LIN {X 95.616,Y 104.988,Z 83.161,A 180.000,B 0.000,C 180.000} C_DIS
LIN {X 95.371,Y 104.988,Z 83.026,A 180.000,B 0.000,C 180.000} C_DIS
LIN {X 94.812,Y 104.988,Z 82.658,A 180.000,B 0.000,C 180.000} C_DIS
LIN {X 94.419,Y 104.988,Z 82.358,A 180.000,B 0.000,C 180.000} C_DIS
LIN {X 93.998,Y 104.988,Z 81.987,A 180.000,B 0.000,C 180.000} C_DIS
LIN {X 93.703,Y 104.988,Z 81.713,A 180.000,B 0.000,C 180.000} C_DIS
LIN {X 93.333,Y 104.988,Z 81.344,A 180.000,B 0.000,C 180.000} C_DIS
LIN {X 92.872,Y 104.988,Z 80.840,A 180.000,B 0.000,C 180.000} C_DIS
LIN {X 92.497,Y 104.988,Z 80.403,A 180.000,B 0.000,C 180.000} C_DIS
LIN {X 92.120,Y 104.988,Z 79.949,A 180.000,B 0.000,C 180.000} C_DIS
LIN {X 91.570,Y 104.988,Z 79.235,A 180.000,B 0.000,C 180.000} C_DIS
LIN {X 90.776,Y 104.988,Z 78.140,A 180.000,B 0.000,C 180.000} C_DIS
LIN {X 90.026,Y 104.988,Z 77.033,A 180.000,B 0.000,C 180.000} C_DIS
LIN {X 89.022,Y 104.988,Z 75.463,A 180.000,B 0.000,C 180.000} C_DIS
LIN {X 88.077,Y 104.988,Z 73.911,A 180.000,B 0.000,C 180.000} C_DIS
LIN {X 86.884,Y 104.988,Z 71.862,A 180.000,B 0.000,C 180.000} C_DIS
LIN {X 85.520,Y 104.988,Z 69.426,A 180.000,B 0.000,C 180.000} C_DIS
LIN {X 84.508,Y 104.988,Z 67.555,A 180.000,B 0.000,C 180.000} C_DIS
LIN {X 84.508,Y 104.988,Z 62.000,A 180.000,B 0.000,C 180.000} C_DIS
LIN {X 70.550,Y 104.988,Z 62.000,A 180.000,B 0.000,C 180.000} C_DIS
LIN {X 70.550,Y 104.988,Z 66.500,A 180.000,B 0.000,C 180.000} C_DIS
LIN {X 70.498,Y 104.988,Z 66.500,A 180.000,B 0.000,C 180.000} C_DIS
LIN {X 70.498,Y 104.988,Z 70.000,A 180.000,B 0.000,C 180.000} C_DIS
LIN {X 65.196,Y 104.988,Z 70.000,A 180.000,B 0.000,C 180.000} C_DIS
LIN {X 65.195,Y 104.988,Z 74.500,A 180.000,B 0.000,C 180.000} C_DIS
LIN {X 65.139,Y 104.988,Z 74.500,A 180.000,B 0.000,C 180.000} C_DIS
LIN {X 65.139,Y 104.988,Z 78.000,A 180.000,B 0.000,C 180.000} C_DIS
LIN {X 51.866,Y 104.988,Z 78.000,A 180.000,B 0.000,C 180.000} C_DIS
LIN {X 51.866,Y 104.988,Z 74.500,A 180.000,B 0.000,C 180.000} C_DIS
LIN {X 51.810,Y 104.988,Z 74.500,A 180.000,B 0.000,C 180.000} C_DIS
LIN {X 51.809,Y 104.988,Z 70.000,A 180.000,B 0.000,C 180.000} C_DIS
LIN {X 46.502,Y 104.988,Z 70.000,A 180.000,B 0.000,C 180.000} C_DIS
LIN {X 46.499,Y 104.988,Z 66.500,A 180.000,B 0.000,C 180.000} C_DIS
LIN {X 46.450,Y 104.988,Z 66.500,A 180.000,B 0.000,C 180.000} C_DIS
LIN {X 46.450,Y 104.988,Z 62.000,A 180.000,B 0.000,C 180.000} C_DIS
LIN {X 36.453,Y 104.988,Z 62.000,A 180.000,B 0.000,C 180.000} C_DIS
LIN {X 36.453,Y 104.988,Z 57.000,A 180.000,B 0.000,C 180.000} C_DIS
LIN {X 7.719,Y 104.988,Z 57.000,A 180.000,B 0.000,C 180.000} C_DIS
LIN {X 7.719,Y 104.988,Z 52.000,A 180.000,B 0.000,C 180.000} C_DIS
LIN {X 2.500,Y 104.988,Z 52.000,A 180.000,B 0.000,C 180.000} C_DIS
LIN {X 2.500,Y 104.988,Z 45.000,A 180.000,B 0.000,C 180.000} C_DIS
LIN {X -0.010,Y 104.988,Z 45.000,A 180.000,B 0.000,C 180.000} C_DIS
; Link Move Starts
LIN {X -0.120,Y 104.988,Z 45.026,A 180.000,B 0.000,C 180.000} C_DIS
LIN {X -0.230,Y 104.988,Z 45.051,A 180.000,B 0.000,C 180.000} C_DIS
LIN {X -0.771,Y 105.301,Z 45.051,A 180.000,B 0.000,C 180.000} C_DIS
LIN {X -0.771,Y 105.926,Z 45.051,A 180.000,B 0.000,C 180.000} C_DIS
LIN {X -0.230,Y 106.238,Z 45.051,A 180.000,B 0.000,C 180.000} C_DIS
LIN {X -0.120,Y 106.238,Z 45.026,A 180.000,B 0.000,C 180.000} C_DIS
LIN {X -0.010,Y 106.238,Z 45.000,A 180.000,B 0.000,C 180.000} C_DIS
; Cutting Move Starts
LIN {X 2.500,Y 106.238,Z 45.000,A 180.000,B 0.000,C 180.000} C_DIS
LIN {X 2.500,Y 106.238,Z 52.000,A 180.000,B 0.000,C 180.000} C_DIS
LIN {X 8.224,Y 106.238,Z 52.000,A 180.000,B 0.000,C 180.000} C_DIS
LIN {X 8.228,Y 106.238,Z 57.000,A 180.000,B 0.000,C 180.000} C_DIS
LIN {X 37.703,Y 106.238,Z 57.000,A 180.000,B 0.000,C 180.000} C_DIS
LIN {X 37.703,Y 106.238,Z 62.000,A 180.000,B 0.000,C 180.000} C_DIS
LIN {X 46.881,Y 106.238,Z 62.000,A 180.000,B 0.000,C 180.000} C_DIS
LIN {X 46.881,Y 106.238,Z 66.500,A 180.000,B 0.000,C 180.000} C_DIS
LIN {X 46.935,Y 106.238,Z 66.500,A 180.000,B 0.000,C 180.000} C_DIS
LIN {X 46.936,Y 106.238,Z 70.000,A 180.000,B 0.000,C 180.000} C_DIS
LIN {X 52.627,Y 106.238,Z 70.000,A 180.000,B 0.000,C 180.000} C_DIS
LIN {X 52.627,Y 106.238,Z 74.500,A 180.000,B 0.000,C 180.000} C_DIS
LIN {X 52.691,Y 106.238,Z 74.500,A 180.000,B 0.000,C 180.000} C_DIS
LIN {X 52.691,Y 106.238,Z 78.000,A 180.000,B 0.000,C 180.000} C_DIS
LIN {X 64.310,Y 106.238,Z 78.000,A 180.000,B 0.000,C 180.000} C_DIS
LIN {X 64.310,Y 106.238,Z 74.500,A 180.000,B 0.000,C 180.000} C_DIS
LIN {X 64.371,Y 106.238,Z 74.500,A 180.000,B 0.000,C 180.000} C_DIS
LIN {X 64.376,Y 106.238,Z 70.000,A 180.000,B 0.000,C 180.000} C_DIS
LIN {X 70.063,Y 106.238,Z 70.000,A 180.000,B 0.000,C 180.000} C_DIS
LIN {X 70.064,Y 106.238,Z 66.500,A 180.000,B 0.000,C 180.000} C_DIS
LIN {X 70.119,Y 106.238,Z 66.500,A 180.000,B 0.000,C 180.000} C_DIS
LIN {X 70.119,Y 106.238,Z 62.000,A 180.000,B 0.000,C 180.000} C_DIS
LIN {X 85.309,Y 106.238,Z 62.000,A 180.000,B 0.000,C 180.000} C_DIS
LIN {X 85.309,Y 106.238,Z 67.555,A 180.000,B 0.000,C 180.000} C_DIS
LIN {X 86.499,Y 106.238,Z 69.593,A 180.000,B 0.000,C 180.000} C_DIS
LIN {X 87.652,Y 106.238,Z 71.487,A 180.000,B 0.000,C 180.000} C_DIS
LIN {X 88.751,Y 106.238,Z 73.204,A 180.000,B 0.000,C 180.000} C_DIS
LIN {X 89.638,Y 106.238,Z 74.514,A 180.000,B 0.000,C 180.000} C_DIS
LIN {X 90.553,Y 106.238,Z 75.781,A 180.000,B 0.000,C 180.000} C_DIS
LIN {X 91.246,Y 106.238,Z 76.678,A 180.000,B 0.000,C 180.000} C_DIS
LIN {X 91.704,Y 106.238,Z 77.229,A 180.000,B 0.000,C 180.000} C_DIS
LIN {X 92.068,Y 106.238,Z 77.653,A 180.000,B 0.000,C 180.000} C_DIS
LIN {X 92.647,Y 106.238,Z 78.287,A 180.000,B 0.000,C 180.000} C_DIS
LIN {X 93.102,Y 106.238,Z 78.739,A 180.000,B 0.000,C 180.000} C_DIS
LIN {X 93.353,Y 106.238,Z 78.974,A 180.000,B 0.000,C 180.000} C_DIS
LIN {X 93.850,Y 106.238,Z 79.413,A 180.000,B 0.000,C 180.000} C_DIS
LIN {X 94.082,Y 106.238,Z 79.596,A 180.000,B 0.000,C 180.000} C_DIS
LIN {X 94.407,Y 106.238,Z 79.842,A 180.000,B 0.000,C 180.000} C_DIS
LIN {X 95.017,Y 106.238,Z 80.240,A 180.000,B 0.000,C 180.000} C_DIS
LIN {X 95.429,Y 106.238,Z 80.463,A 180.000,B 0.000,C 180.000} C_DIS
LIN {X 95.636,Y 106.238,Z 80.555,A 180.000,B 0.000,C 180.000} C_DIS
LIN {X 96.080,Y 106.238,Z 80.735,A 180.000,B 0.000,C 180.000} C_DIS
LIN {X 96.484,Y 106.238,Z 80.857,A 180.000,B 0.000,C 180.000} C_DIS
LIN {X 96.776,Y 106.238,Z 80.912,A 180.000,B 0.000,C 180.000} C_DIS
LIN {X 97.029,Y 106.238,Z 80.950,A 180.000,B 0.000,C 180.000} C_DIS
LIN {X 97.255,Y 106.238,Z 80.971,A 180.000,B 0.000,C 180.000} C_DIS
LIN {X 97.526,Y 106.238,Z 80.983,A 180.000,B 0.000,C 180.000} C_DIS
LIN {X 97.834,Y 106.238,Z 80.966,A 180.000,B 0.000,C 180.000} C_DIS
LIN {X 98.107,Y 106.238,Z 80.932,A 180.000,B 0.000,C 180.000} C_DIS
LIN {X 98.493,Y 106.238,Z 80.862,A 180.000,B 0.000,C 180.000} C_DIS
LIN {X 98.803,Y 106.238,Z 80.772,A 180.000,B 0.000,C 180.000} C_DIS
LIN {X 98.999,Y 106.238,Z 80.704,A 180.000,B 0.000,C 180.000} C_DIS
LIN {X 99.513,Y 106.238,Z 80.491,A 180.000,B 0.000,C 180.000} C_DIS
LIN {X 99.761,Y 106.238,Z 80.362,A 180.000,B 0.000,C 180.000} C_DIS
LIN {X 100.001,Y 106.238,Z 80.229,A 180.000,B 0.000,C 180.000} C_DIS
LIN {X 100.606,Y 106.238,Z 79.832,A 180.000,B 0.000,C 180.000} C_DIS
LIN {X 101.068,Y 106.238,Z 79.481,A 180.000,B 0.000,C 180.000} C_DIS
LIN {X 101.407,Y 106.238,Z 79.188,A 180.000,B 0.000,C 180.000} C_DIS
LIN {X 101.768,Y 106.238,Z 78.864,A 180.000,B 0.000,C 180.000} C_DIS
LIN {X 102.297,Y 106.238,Z 78.345,A 180.000,B 0.000,C 180.000} C_DIS
LIN {X 102.749,Y 106.238,Z 77.856,A 180.000,B 0.000,C 180.000} C_DIS
LIN {X 103.049,Y 106.238,Z 77.520,A 180.000,B 0.000,C 180.000} C_DIS
LIN {X 103.690,Y 106.238,Z 76.757,A 180.000,B 0.000,C 180.000} C_DIS
LIN {X 104.418,Y 106.238,Z 75.820,A 180.000,B 0.000,C 180.000} C_DIS
LIN {X 105.298,Y 106.238,Z 74.605,A 180.000,B 0.000,C 180.000} C_DIS
LIN {X 106.168,Y 106.238,Z 73.327,A 180.000,B 0.000,C 180.000} C_DIS
LIN {X 107.258,Y 106.238,Z 71.631,A 180.000,B 0.000,C 180.000} C_DIS
LIN {X 108.395,Y 106.238,Z 69.771,A 180.000,B 0.000,C 180.000} C_DIS
LIN {X 109.689,Y 106.238,Z 67.558,A 180.000,B 0.000,C 180.000} C_DIS
LIN {X 109.691,Y 106.238,Z 62.000,A 180.000,B 0.000,C 180.000} C_DIS
LIN {X 117.295,Y 106.238,Z 62.000,A 180.000,B 0.000,C 180.000} C_DIS
LIN {X 117.297,Y 106.238,Z 57.000,A 180.000,B 0.000,C 180.000} C_DIS
LIN {X 146.772,Y 106.238,Z 57.000,A 180.000,B 0.000,C 180.000} C_DIS
LIN {X 146.772,Y 106.238,Z 52.000,A 180.000,B 0.000,C 180.000} C_DIS
LIN {X 152.500,Y 106.238,Z 52.000,A 180.000,B 0.000,C 180.000} C_DIS
LIN {X 152.500,Y 106.238,Z 45.000,A 180.000,B 0.000,C 180.000} C_DIS
LIN {X 155.010,Y 106.238,Z 45.000,A 180.000,B 0.000,C 180.000} C_DIS
; Link Move Starts
LIN {X 155.120,Y 106.238,Z 45.026,A 180.000,B 0.000,C 180.000} C_DIS
LIN {X 155.230,Y 106.238,Z 45.051,A 180.000,B 0.000,C 180.000} C_DIS
LIN {X 155.771,Y 106.551,Z 45.051,A 180.000,B 0.000,C 180.000} C_DIS
LIN {X 155.771,Y 107.176,Z 45.051,A 180.000,B 0.000,C 180.000} C_DIS
LIN {X 155.230,Y 107.488,Z 45.051,A 180.000,B 0.000,C 180.000} C_DIS
LIN {X 155.120,Y 107.488,Z 45.026,A 180.000,B 0.000,C 180.000} C_DIS
LIN {X 155.010,Y 107.488,Z 45.000,A 180.000,B 0.000,C 180.000} C_DIS
; Cutting Move Starts
LIN {X 152.500,Y 107.488,Z 45.000,A 180.000,B 0.000,C 180.000} C_DIS
LIN {X 152.500,Y 107.488,Z 52.000,A 180.000,B 0.000,C 180.000} C_DIS
LIN {X 146.238,Y 107.488,Z 52.000,A 180.000,B 0.000,C 180.000} C_DIS
LIN {X 146.238,Y 107.488,Z 57.000,A 180.000,B 0.000,C 180.000} C_DIS
LIN {X 116.047,Y 107.488,Z 57.000,A 180.000,B 0.000,C 180.000} C_DIS
LIN {X 116.047,Y 107.488,Z 62.000,A 180.000,B 0.000,C 180.000} C_DIS
LIN {X 108.691,Y 107.488,Z 62.000,A 180.000,B 0.000,C 180.000} C_DIS
LIN {X 108.688,Y 107.488,Z 67.559,A 180.000,B 0.000,C 180.000} C_DIS
LIN {X 107.443,Y 107.488,Z 69.499,A 180.000,B 0.000,C 180.000} C_DIS
LIN {X 106.403,Y 107.488,Z 71.028,A 180.000,B 0.000,C 180.000} C_DIS
LIN {X 105.423,Y 107.488,Z 72.382,A 180.000,B 0.000,C 180.000} C_DIS
LIN {X 104.570,Y 107.488,Z 73.479,A 180.000,B 0.000,C 180.000} C_DIS
LIN {X 103.804,Y 107.488,Z 74.390,A 180.000,B 0.000,C 180.000} C_DIS
LIN {X 103.504,Y 107.488,Z 74.725,A 180.000,B 0.000,C 180.000} C_DIS
LIN {X 102.991,Y 107.488,Z 75.279,A 180.000,B 0.000,C 180.000} C_DIS
LIN {X 102.351,Y 107.488,Z 75.907,A 180.000,B 0.000,C 180.000} C_DIS
LIN {X 102.000,Y 107.488,Z 76.221,A 180.000,B 0.000,C 180.000} C_DIS
LIN {X 101.597,Y 107.488,Z 76.571,A 180.000,B 0.000,C 180.000} C_DIS
LIN {X 101.032,Y 107.488,Z 77.002,A 180.000,B 0.000,C 180.000} C_DIS
LIN {X 100.369,Y 107.488,Z 77.435,A 180.000,B 0.000,C 180.000} C_DIS
LIN {X 100.126,Y 107.488,Z 77.570,A 180.000,B 0.000,C 180.000} C_DIS
LIN {X 99.798,Y 107.488,Z 77.742,A 180.000,B 0.000,C 180.000} C_DIS
LIN {X 99.210,Y 107.488,Z 77.987,A 180.000,B 0.000,C 180.000} C_DIS
LIN {X 99.019,Y 107.488,Z 78.052,A 180.000,B 0.000,C 180.000} C_DIS
LIN {X 98.633,Y 107.488,Z 78.165,A 180.000,B 0.000,C 180.000} C_DIS
LIN {X 98.157,Y 107.488,Z 78.251,A 180.000,B 0.000,C 180.000} C_DIS
LIN {X 97.920,Y 107.488,Z 78.280,A 180.000,B 0.000,C 180.000} C_DIS
LIN {X 97.529,Y 107.488,Z 78.303,A 180.000,B 0.000,C 180.000} C_DIS
LIN {X 97.268,Y 107.488,Z 78.291,A 180.000,B 0.000,C 180.000} C_DIS
LIN {X 96.984,Y 107.488,Z 78.270,A 180.000,B 0.000,C 180.000} C_DIS
LIN {X 96.715,Y 107.488,Z 78.230,A 180.000,B 0.000,C 180.000} C_DIS
LIN {X 96.353,Y 107.488,Z 78.162,A 180.000,B 0.000,C 180.000} C_DIS
LIN {X 95.857,Y 107.488,Z 78.013,A 180.000,B 0.000,C 180.000} C_DIS
LIN {X 95.438,Y 107.488,Z 77.842,A 180.000,B 0.000,C 180.000} C_DIS
LIN {X 95.169,Y 107.488,Z 77.727,A 180.000,B 0.000,C 180.000} C_DIS
LIN {X 94.651,Y 107.488,Z 77.448,A 180.000,B 0.000,C 180.000} C_DIS
LIN {X 93.979,Y 107.488,Z 77.009,A 180.000,B 0.000,C 180.000} C_DIS
LIN {X 93.591,Y 107.488,Z 76.716,A 180.000,B 0.000,C 180.000} C_DIS
LIN {X 93.340,Y 107.488,Z 76.518,A 180.000,B 0.000,C 180.000} C_DIS
LIN {X 92.731,Y 107.488,Z 75.982,A 180.000,B 0.000,C 180.000} C_DIS
LIN {X 92.465,Y 107.488,Z 75.730,A 180.000,B 0.000,C 180.000} C_DIS
LIN {X 91.957,Y 107.488,Z 75.226,A 180.000,B 0.000,C 180.000} C_DIS
LIN {X 91.256,Y 107.488,Z 74.459,A 180.000,B 0.000,C 180.000} C_DIS
LIN {X 90.882,Y 107.488,Z 74.020,A 180.000,B 0.000,C 180.000} C_DIS
LIN {X 90.370,Y 107.488,Z 73.405,A 180.000,B 0.000,C 180.000} C_DIS
LIN {X 89.537,Y 107.488,Z 72.327,A 180.000,B 0.000,C 180.000} C_DIS
LIN {X 88.532,Y 107.488,Z 70.935,A 180.000,B 0.000,C 180.000} C_DIS
LIN {X 87.483,Y 107.488,Z 69.386,A 180.000,B 0.000,C 180.000} C_DIS
LIN {X 86.309,Y 107.488,Z 67.555,A 180.000,B 0.000,C 180.000} C_DIS
LIN {X 86.308,Y 107.488,Z 62.000,A 180.000,B 0.000,C 180.000} C_DIS
LIN {X 69.529,Y 107.488,Z 62.000,A 180.000,B 0.000,C 180.000} C_DIS
LIN {X 69.528,Y 107.488,Z 66.500,A 180.000,B 0.000,C 180.000} C_DIS
LIN {X 69.472,Y 107.488,Z 66.500,A 180.000,B 0.000,C 180.000} C_DIS
LIN {X 69.471,Y 107.488,Z 70.000,A 180.000,B 0.000,C 180.000} C_DIS
LIN {X 63.096,Y 107.488,Z 70.000,A 180.000,B 0.000,C 180.000} C_DIS
LIN {X 63.096,Y 107.488,Z 74.500,A 180.000,B 0.000,C 180.000} C_DIS
LIN {X 63.016,Y 107.488,Z 74.500,A 180.000,B 0.000,C 180.000} C_DIS
LIN {X 63.014,Y 107.488,Z 78.000,A 180.000,B 0.000,C 180.000} C_DIS
LIN {X 53.992,Y 107.488,Z 78.000,A 180.000,B 0.000,C 180.000} C_DIS
LIN {X 53.992,Y 107.488,Z 74.500,A 180.000,B 0.000,C 180.000} C_DIS
LIN {X 53.909,Y 107.488,Z 74.500,A 180.000,B 0.000,C 180.000} C_DIS
LIN {X 53.909,Y 107.488,Z 70.000,A 180.000,B 0.000,C 180.000} C_DIS
LIN {X 47.528,Y 107.488,Z 70.000,A 180.000,B 0.000,C 180.000} C_DIS
LIN {X 47.527,Y 107.488,Z 66.500,A 180.000,B 0.000,C 180.000} C_DIS
LIN {X 47.471,Y 107.488,Z 66.500,A 180.000,B 0.000,C 180.000} C_DIS
LIN {X 47.471,Y 107.488,Z 62.000,A 180.000,B 0.000,C 180.000} C_DIS
LIN {X 38.953,Y 107.488,Z 62.000,A 180.000,B 0.000,C 180.000} C_DIS
LIN {X 38.952,Y 107.488,Z 57.000,A 180.000,B 0.000,C 180.000} C_DIS
LIN {X 8.762,Y 107.488,Z 57.000,A 180.000,B 0.000,C 180.000} C_DIS
LIN {X 8.762,Y 107.488,Z 52.000,A 180.000,B 0.000,C 180.000} C_DIS
LIN {X 2.500,Y 107.488,Z 52.000,A 180.000,B 0.000,C 180.000} C_DIS
LIN {X 2.500,Y 107.488,Z 45.000,A 180.000,B 0.000,C 180.000} C_DIS
LIN {X -0.010,Y 107.488,Z 45.000,A 180.000,B 0.000,C 180.000} C_DIS
; Link Move Starts
LIN {X -0.120,Y 107.488,Z 45.026,A 180.000,B 0.000,C 180.000} C_DIS
LIN {X -0.230,Y 107.488,Z 45.051,A 180.000,B 0.000,C 180.000} C_DIS
LIN {X -0.771,Y 107.801,Z 45.051,A 180.000,B 0.000,C 180.000} C_DIS
LIN {X -0.771,Y 108.425,Z 45.051,A 180.000,B 0.000,C 180.000} C_DIS
LIN {X -0.230,Y 108.738,Z 45.051,A 180.000,B 0.000,C 180.000} C_DIS
LIN {X -0.120,Y 108.738,Z 45.026,A 180.000,B 0.000,C 180.000} C_DIS
LIN {X -0.010,Y 108.738,Z 45.000,A 180.000,B 0.000,C 180.000} C_DIS
; Cutting Move Starts
LIN {X 2.500,Y 108.738,Z 45.000,A 180.000,B 0.000,C 180.000} C_DIS
LIN {X 2.500,Y 108.738,Z 52.000,A 180.000,B 0.000,C 180.000} C_DIS
LIN {X 9.316,Y 108.738,Z 52.000,A 180.000,B 0.000,C 180.000} C_DIS
LIN {X 9.320,Y 108.738,Z 57.000,A 180.000,B 0.000,C 180.000} C_DIS
LIN {X 40.202,Y 108.738,Z 57.000,A 180.000,B 0.000,C 180.000} C_DIS
LIN {X 40.202,Y 108.738,Z 62.000,A 180.000,B 0.000,C 180.000} C_DIS
LIN {X 48.247,Y 108.738,Z 62.000,A 180.000,B 0.000,C 180.000} C_DIS
LIN {X 48.251,Y 108.738,Z 66.500,A 180.000,B 0.000,C 180.000} C_DIS
LIN {X 48.311,Y 108.738,Z 66.500,A 180.000,B 0.000,C 180.000} C_DIS
LIN {X 48.311,Y 108.738,Z 70.000,A 180.000,B 0.000,C 180.000} C_DIS
LIN {X 56.369,Y 108.738,Z 70.000,A 180.000,B 0.000,C 180.000} C_DIS
LIN {X 56.369,Y 108.738,Z 74.500,A 180.000,B 0.000,C 180.000} C_DIS
LIN {X 56.545,Y 108.738,Z 74.500,A 180.000,B 0.000,C 180.000} C_DIS
LIN {X 56.545,Y 108.738,Z 78.000,A 180.000,B 0.000,C 180.000} C_DIS
LIN {X 60.452,Y 108.738,Z 78.000,A 180.000,B 0.000,C 180.000} C_DIS
LIN {X 60.452,Y 108.738,Z 74.500,A 180.000,B 0.000,C 180.000} C_DIS
LIN {X 60.648,Y 108.738,Z 74.500,A 180.000,B 0.000,C 180.000} C_DIS
LIN {X 60.648,Y 108.738,Z 70.000,A 180.000,B 0.000,C 180.000} C_DIS
LIN {X 68.685,Y 108.738,Z 70.000,A 180.000,B 0.000,C 180.000} C_DIS
LIN {X 68.689,Y 108.738,Z 66.500,A 180.000,B 0.000,C 180.000} C_DIS
LIN {X 68.749,Y 108.738,Z 66.500,A 180.000,B 0.000,C 180.000} C_DIS
LIN {X 68.749,Y 108.738,Z 62.000,A 180.000,B 0.000,C 180.000} C_DIS
LIN {X 87.566,Y 108.738,Z 62.000,A 180.000,B 0.000,C 180.000} C_DIS
LIN {X 87.566,Y 108.738,Z 67.555,A 180.000,B 0.000,C 180.000} C_DIS
LIN {X 88.517,Y 108.738,Z 68.869,A 180.000,B 0.000,C 180.000} C_DIS
LIN {X 89.472,Y 108.738,Z 70.105,A 180.000,B 0.000,C 180.000} C_DIS
LIN {X 89.816,Y 108.738,Z 70.520,A 180.000,B 0.000,C 180.000} C_DIS
LIN {X 90.450,Y 108.738,Z 71.272,A 180.000,B 0.000,C 180.000} C_DIS
LIN {X 91.276,Y 108.738,Z 72.173,A 180.000,B 0.000,C 180.000} C_DIS
LIN {X 92.056,Y 108.738,Z 72.942,A 180.000,B 0.000,C 180.000} C_DIS
LIN {X 92.410,Y 108.738,Z 73.257,A 180.000,B 0.000,C 180.000} C_DIS
LIN {X 92.879,Y 108.738,Z 73.664,A 180.000,B 0.000,C 180.000} C_DIS
LIN {X 93.546,Y 108.738,Z 74.173,A 180.000,B 0.000,C 180.000} C_DIS
LIN {X 94.282,Y 108.738,Z 74.653,A 180.000,B 0.000,C 180.000} C_DIS
LIN {X 94.896,Y 108.738,Z 74.984,A 180.000,B 0.000,C 180.000} C_DIS
LIN {X 95.231,Y 108.738,Z 75.127,A 180.000,B 0.000,C 180.000} C_DIS
LIN {X 95.631,Y 108.738,Z 75.290,A 180.000,B 0.000,C 180.000} C_DIS
LIN {X 96.220,Y 108.738,Z 75.467,A 180.000,B 0.000,C 180.000} C_DIS
LIN {X 96.675,Y 108.738,Z 75.551,A 180.000,B 0.000,C 180.000} C_DIS
LIN {X 96.914,Y 108.738,Z 75.587,A 180.000,B 0.000,C 180.000} C_DIS
LIN {X 97.296,Y 108.738,Z 75.613,A 180.000,B 0.000,C 180.000} C_DIS
LIN {X 97.537,Y 108.738,Z 75.622,A 180.000,B 0.000,C 180.000} C_DIS
LIN {X 98.004,Y 108.738,Z 75.594,A 180.000,B 0.000,C 180.000} C_DIS
LIN {X 98.208,Y 108.738,Z 75.571,A 180.000,B 0.000,C 180.000} C_DIS
LIN {X 98.773,Y 108.738,Z 75.468,A 180.000,B 0.000,C 180.000} C_DIS
LIN {X 99.123,Y 108.738,Z 75.366,A 180.000,B 0.000,C 180.000} C_DIS
LIN {X 99.388,Y 108.738,Z 75.283,A 180.000,B 0.000,C 180.000} C_DIS
LIN {X 99.965,Y 108.738,Z 75.045,A 180.000,B 0.000,C 180.000} C_DIS
LIN {X 100.174,Y 108.738,Z 74.947,A 180.000,B 0.000,C 180.000} C_DIS
LIN {X 100.723,Y 108.738,Z 74.650,A 180.000,B 0.000,C 180.000} C_DIS
LIN {X 101.455,Y 108.738,Z 74.173,A 180.000,B 0.000,C 180.000} C_DIS
LIN {X 102.121,Y 108.738,Z 73.664,A 180.000,B 0.000,C 180.000} C_DIS
LIN {X 102.549,Y 108.738,Z 73.293,A 180.000,B 0.000,C 180.000} C_DIS
LIN {X 102.932,Y 108.738,Z 72.953,A 180.000,B 0.000,C 180.000} C_DIS
LIN {X 103.673,Y 108.738,Z 72.226,A 180.000,B 0.000,C 180.000} C_DIS
LIN {X 104.030,Y 108.738,Z 71.841,A 180.000,B 0.000,C 180.000} C_DIS
LIN {X 104.563,Y 108.738,Z 71.256,A 180.000,B 0.000,C 180.000} C_DIS
LIN {X 105.451,Y 108.738,Z 70.201,A 180.000,B 0.000,C 180.000} C_DIS
LIN {X 106.426,Y 108.738,Z 68.945,A 180.000,B 0.000,C 180.000} C_DIS
LIN {X 107.434,Y 108.738,Z 67.555,A 180.000,B 0.000,C 180.000} C_DIS
LIN {X 107.434,Y 108.738,Z 62.000,A 180.000,B 0.000,C 180.000} C_DIS
LIN {X 114.795,Y 108.738,Z 62.000,A 180.000,B 0.000,C 180.000} C_DIS
LIN {X 114.798,Y 108.738,Z 57.000,A 180.000,B 0.000,C 180.000} C_DIS
LIN {X 145.680,Y 108.738,Z 57.000,A 180.000,B 0.000,C 180.000} C_DIS
LIN {X 145.680,Y 108.738,Z 52.000,A 180.000,B 0.000,C 180.000} C_DIS
LIN {X 152.500,Y 108.738,Z 52.000,A 180.000,B 0.000,C 180.000} C_DIS
LIN {X 152.500,Y 108.738,Z 45.000,A 180.000,B 0.000,C 180.000} C_DIS
LIN {X 155.010,Y 108.738,Z 45.000,A 180.000,B 0.000,C 180.000} C_DIS
; Link Move Starts
LIN {X 155.120,Y 108.738,Z 45.026,A 180.000,B 0.000,C 180.000} C_DIS
LIN {X 155.230,Y 108.738,Z 45.051,A 180.000,B 0.000,C 180.000} C_DIS
LIN {X 155.771,Y 109.050,Z 45.051,A 180.000,B 0.000,C 180.000} C_DIS
LIN {X 155.771,Y 109.675,Z 45.051,A 180.000,B 0.000,C 180.000} C_DIS
LIN {X 155.230,Y 109.988,Z 45.051,A 180.000,B 0.000,C 180.000} C_DIS
LIN {X 155.120,Y 109.988,Z 45.026,A 180.000,B 0.000,C 180.000} C_DIS
LIN {X 155.010,Y 109.988,Z 45.000,A 180.000,B 0.000,C 180.000} C_DIS
; Cutting Move Starts
LIN {X 152.500,Y 109.988,Z 45.000,A 180.000,B 0.000,C 180.000} C_DIS
LIN {X 152.500,Y 109.988,Z 52.000,A 180.000,B 0.000,C 180.000} C_DIS
LIN {X 145.096,Y 109.988,Z 52.000,A 180.000,B 0.000,C 180.000} C_DIS
LIN {X 145.093,Y 109.988,Z 57.000,A 180.000,B 0.000,C 180.000} C_DIS
LIN {X 113.548,Y 109.988,Z 57.000,A 180.000,B 0.000,C 180.000} C_DIS
LIN {X 113.548,Y 109.988,Z 62.000,A 180.000,B 0.000,C 180.000} C_DIS
LIN {X 105.801,Y 109.988,Z 62.000,A 180.000,B 0.000,C 180.000} C_DIS
LIN {X 105.801,Y 109.988,Z 67.555,A 180.000,B 0.000,C 180.000} C_DIS
LIN {X 105.313,Y 109.988,Z 68.132,A 180.000,B 0.000,C 180.000} C_DIS
LIN {X 104.382,Y 109.988,Z 69.144,A 180.000,B 0.000,C 180.000} C_DIS
LIN {X 103.516,Y 109.988,Z 69.996,A 180.000,B 0.000,C 180.000} C_DIS
LIN {X 102.669,Y 109.988,Z 70.739,A 180.000,B 0.000,C 180.000} C_DIS
LIN {X 101.880,Y 109.988,Z 71.342,A 180.000,B 0.000,C 180.000} C_DIS
LIN {X 101.078,Y 109.988,Z 71.864,A 180.000,B 0.000,C 180.000} C_DIS
LIN {X 100.362,Y 109.988,Z 72.248,A 180.000,B 0.000,C 180.000} C_DIS
LIN {X 99.619,Y 109.988,Z 72.558,A 180.000,B 0.000,C 180.000} C_DIS
LIN {X 99.375,Y 109.988,Z 72.635,A 180.000,B 0.000,C 180.000} C_DIS
LIN {X 98.908,Y 109.988,Z 72.772,A 180.000,B 0.000,C 180.000} C_DIS
LIN {X 98.249,Y 109.988,Z 72.891,A 180.000,B 0.000,C 180.000} C_DIS
LIN {X 98.010,Y 109.988,Z 72.914,A 180.000,B 0.000,C 180.000} C_DIS
LIN {X 97.520,Y 109.988,Z 72.942,A 180.000,B 0.000,C 180.000} C_DIS
LIN {X 97.112,Y 109.988,Z 72.921,A 180.000,B 0.000,C 180.000} C_DIS
LIN {X 96.821,Y 109.988,Z 72.901,A 180.000,B 0.000,C 180.000} C_DIS
LIN {X 96.564,Y 109.988,Z 72.859,A 180.000,B 0.000,C 180.000} C_DIS
LIN {X 96.079,Y 109.988,Z 72.769,A 180.000,B 0.000,C 180.000} C_DIS
LIN {X 95.404,Y 109.988,Z 72.566,A 180.000,B 0.000,C 180.000} C_DIS
LIN {X 94.956,Y 109.988,Z 72.383,A 180.000,B 0.000,C 180.000} C_DIS
LIN {X 94.621,Y 109.988,Z 72.240,A 180.000,B 0.000,C 180.000} C_DIS
LIN {X 93.913,Y 109.988,Z 71.859,A 180.000,B 0.000,C 180.000} C_DIS
LIN {X 93.117,Y 109.988,Z 71.340,A 180.000,B 0.000,C 180.000} C_DIS
LIN {X 92.327,Y 109.988,Z 70.735,A 180.000,B 0.000,C 180.000} C_DIS
LIN {X 91.485,Y 109.988,Z 69.997,A 180.000,B 0.000,C 180.000} C_DIS
LIN {X 90.610,Y 109.988,Z 69.137,A 180.000,B 0.000,C 180.000} C_DIS
LIN {X 89.643,Y 109.988,Z 68.082,A 180.000,B 0.000,C 180.000} C_DIS
LIN {X 89.199,Y 109.988,Z 67.555,A 180.000,B 0.000,C 180.000} C_DIS
LIN {X 89.198,Y 109.988,Z 62.000,A 180.000,B 0.000,C 180.000} C_DIS
LIN {X 67.741,Y 109.988,Z 62.000,A 180.000,B 0.000,C 180.000} C_DIS
LIN {X 67.741,Y 109.988,Z 66.500,A 180.000,B 0.000,C 180.000} C_DIS
LIN {X 67.675,Y 109.988,Z 66.500,A 180.000,B 0.000,C 180.000} C_DIS
LIN {X 67.675,Y 109.988,Z 70.000,A 180.000,B 0.000,C 180.000} C_DIS
LIN {X 49.325,Y 109.988,Z 70.000,A 180.000,B 0.000,C 180.000} C_DIS
LIN {X 49.324,Y 109.988,Z 66.500,A 180.000,B 0.000,C 180.000} C_DIS
LIN {X 49.259,Y 109.988,Z 66.500,A 180.000,B 0.000,C 180.000} C_DIS
LIN {X 49.259,Y 109.988,Z 62.000,A 180.000,B 0.000,C 180.000} C_DIS
LIN {X 41.452,Y 109.988,Z 62.000,A 180.000,B 0.000,C 180.000} C_DIS
LIN {X 41.452,Y 109.988,Z 57.000,A 180.000,B 0.000,C 180.000} C_DIS
LIN {X 9.904,Y 109.988,Z 57.000,A 180.000,B 0.000,C 180.000} C_DIS
LIN {X 9.904,Y 109.988,Z 52.000,A 180.000,B 0.000,C 180.000} C_DIS
LIN {X 2.500,Y 109.988,Z 52.000,A 180.000,B 0.000,C 180.000} C_DIS
LIN {X 2.496,Y 109.988,Z 45.000,A 180.000,B 0.000,C 180.000} C_DIS
LIN {X -0.010,Y 109.988,Z 45.000,A 180.000,B 0.000,C 180.000} C_DIS
; Link Move Starts
LIN {X -0.120,Y 109.988,Z 45.026,A 180.000,B 0.000,C 180.000} C_DIS
LIN {X -0.230,Y 109.988,Z 45.051,A 180.000,B 0.000,C 180.000} C_DIS
LIN {X -0.771,Y 110.300,Z 45.051,A 180.000,B 0.000,C 180.000} C_DIS
LIN {X -0.771,Y 110.925,Z 45.051,A 180.000,B 0.000,C 180.000} C_DIS
LIN {X -0.230,Y 111.238,Z 45.051,A 180.000,B 0.000,C 180.000} C_DIS
LIN {X -0.120,Y 111.238,Z 45.026,A 180.000,B 0.000,C 180.000} C_DIS
LIN {X -0.010,Y 111.238,Z 45.000,A 180.000,B 0.000,C 180.000} C_DIS
; Cutting Move Starts
LIN {X 2.499,Y 111.238,Z 45.000,A 180.000,B 0.000,C 180.000} C_DIS
LIN {X 2.500,Y 111.238,Z 52.000,A 180.000,B 0.000,C 180.000} C_DIS
LIN {X 10.519,Y 111.238,Z 52.000,A 180.000,B 0.000,C 180.000} C_DIS
LIN {X 10.519,Y 111.238,Z 57.000,A 180.000,B 0.000,C 180.000} C_DIS
LIN {X 34.632,Y 111.238,Z 57.000,A 180.000,B 0.000,C 180.000} C_DIS
LIN {X 34.632,Y 111.238,Z 52.000,A 180.000,B 0.000,C 180.000} C_DIS
LIN {X 38.368,Y 111.238,Z 52.000,A 180.000,B 0.000,C 180.000} C_DIS
LIN {X 38.368,Y 111.238,Z 57.000,A 180.000,B 0.000,C 180.000} C_DIS
LIN {X 42.702,Y 111.238,Z 57.000,A 180.000,B 0.000,C 180.000} C_DIS
LIN {X 42.702,Y 111.238,Z 62.000,A 180.000,B 0.000,C 180.000} C_DIS
LIN {X 50.586,Y 111.238,Z 62.000,A 180.000,B 0.000,C 180.000} C_DIS
LIN {X 50.586,Y 111.238,Z 66.500,A 180.000,B 0.000,C 180.000} C_DIS
LIN {X 50.667,Y 111.238,Z 66.500,A 180.000,B 0.000,C 180.000} C_DIS
LIN {X 50.667,Y 111.238,Z 70.000,A 180.000,B 0.000,C 180.000} C_DIS
LIN {X 66.333,Y 111.238,Z 70.000,A 180.000,B 0.000,C 180.000} C_DIS
LIN {X 66.333,Y 111.238,Z 66.500,A 180.000,B 0.000,C 180.000} C_DIS
LIN {X 66.414,Y 111.238,Z 66.500,A 180.000,B 0.000,C 180.000} C_DIS
LIN {X 66.414,Y 111.238,Z 62.000,A 180.000,B 0.000,C 180.000} C_DIS
LIN {X 91.484,Y 111.238,Z 62.000,A 180.000,B 0.000,C 180.000} C_DIS
LIN {X 91.488,Y 111.238,Z 67.555,A 180.000,B 0.000,C 180.000} C_DIS
LIN {X 91.801,Y 111.238,Z 67.827,A 180.000,B 0.000,C 180.000} C_DIS
LIN {X 92.685,Y 111.238,Z 68.505,A 180.000,B 0.000,C 180.000} C_DIS
LIN {X 93.540,Y 111.238,Z 69.062,A 180.000,B 0.000,C 180.000} C_DIS
LIN {X 94.286,Y 111.238,Z 69.464,A 180.000,B 0.000,C 180.000} C_DIS
LIN {X 94.488,Y 111.238,Z 69.557,A 180.000,B 0.000,C 180.000} C_DIS
LIN {X 95.178,Y 111.238,Z 69.843,A 180.000,B 0.000,C 180.000} C_DIS
LIN {X 95.945,Y 111.238,Z 70.074,A 180.000,B 0.000,C 180.000} C_DIS
LIN {X 96.447,Y 111.238,Z 70.166,A 180.000,B 0.000,C 180.000} C_DIS
LIN {X 96.741,Y 111.238,Z 70.216,A 180.000,B 0.000,C 180.000} C_DIS
LIN {X 97.246,Y 111.238,Z 70.249,A 180.000,B 0.000,C 180.000} C_DIS
LIN {X 97.535,Y 111.238,Z 70.261,A 180.000,B 0.000,C 180.000} C_DIS
LIN {X 98.122,Y 111.238,Z 70.227,A 180.000,B 0.000,C 180.000} C_DIS
LIN {X 98.304,Y 111.238,Z 70.210,A 180.000,B 0.000,C 180.000} C_DIS
LIN {X 99.044,Y 111.238,Z 70.076,A 180.000,B 0.000,C 180.000} C_DIS
LIN {X 99.338,Y 111.238,Z 69.991,A 180.000,B 0.000,C 180.000} C_DIS
LIN {X 99.830,Y 111.238,Z 69.840,A 180.000,B 0.000,C 180.000} C_DIS
LIN {X 100.638,Y 111.238,Z 69.503,A 180.000,B 0.000,C 180.000} C_DIS
LIN {X 101.447,Y 111.238,Z 69.070,A 180.000,B 0.000,C 180.000} C_DIS
LIN {X 102.302,Y 111.238,Z 68.514,A 180.000,B 0.000,C 180.000} C_DIS
LIN {X 103.143,Y 111.238,Z 67.873,A 180.000,B 0.000,C 180.000} C_DIS
LIN {X 103.508,Y 111.238,Z 67.558,A 180.000,B 0.000,C 180.000} C_DIS
LIN {X 103.512,Y 111.238,Z 62.000,A 180.000,B 0.000,C 180.000} C_DIS
LIN {X 112.298,Y 111.238,Z 62.000,A 180.000,B 0.000,C 180.000} C_DIS
LIN {X 112.298,Y 111.238,Z 57.000,A 180.000,B 0.000,C 180.000} C_DIS
LIN {X 116.632,Y 111.238,Z 57.000,A 180.000,B 0.000,C 180.000} C_DIS
LIN {X 116.632,Y 111.238,Z 52.000,A 180.000,B 0.000,C 180.000} C_DIS
LIN {X 120.368,Y 111.238,Z 52.000,A 180.000,B 0.000,C 180.000} C_DIS
LIN {X 120.368,Y 111.238,Z 57.000,A 180.000,B 0.000,C 180.000} C_DIS
LIN {X 144.480,Y 111.238,Z 57.000,A 180.000,B 0.000,C 180.000} C_DIS
LIN {X 144.481,Y 111.238,Z 52.000,A 180.000,B 0.000,C 180.000} C_DIS
LIN {X 152.500,Y 111.238,Z 52.000,A 180.000,B 0.000,C 180.000} C_DIS
LIN {X 152.500,Y 111.238,Z 45.000,A 180.000,B 0.000,C 180.000} C_DIS
LIN {X 155.010,Y 111.238,Z 45.000,A 180.000,B 0.000,C 180.000} C_DIS
; Link Move Starts
LIN {X 155.120,Y 111.238,Z 45.026,A 180.000,B 0.000,C 180.000} C_DIS
LIN {X 155.230,Y 111.238,Z 45.051,A 180.000,B 0.000,C 180.000} C_DIS
LIN {X 155.771,Y 111.550,Z 45.051,A 180.000,B 0.000,C 180.000} C_DIS
LIN {X 155.771,Y 112.175,Z 45.051,A 180.000,B 0.000,C 180.000} C_DIS
LIN {X 155.230,Y 112.488,Z 45.051,A 180.000,B 0.000,C 180.000} C_DIS
LIN {X 155.120,Y 112.488,Z 45.026,A 180.000,B 0.000,C 180.000} C_DIS
LIN {X 155.010,Y 112.488,Z 45.000,A 180.000,B 0.000,C 180.000} C_DIS
; Cutting Move Starts
LIN {X 152.500,Y 112.488,Z 45.000,A 180.000,B 0.000,C 180.000} C_DIS
LIN {X 152.500,Y 112.488,Z 52.000,A 180.000,B 0.000,C 180.000} C_DIS
LIN {X 143.834,Y 112.488,Z 52.000,A 180.000,B 0.000,C 180.000} C_DIS
LIN {X 143.834,Y 112.488,Z 57.000,A 180.000,B 0.000,C 180.000} C_DIS
LIN {X 122.978,Y 112.488,Z 57.000,A 180.000,B 0.000,C 180.000} C_DIS
LIN {X 122.974,Y 112.488,Z 52.000,A 180.000,B 0.000,C 180.000} C_DIS
LIN {X 114.022,Y 112.488,Z 52.000,A 180.000,B 0.000,C 180.000} C_DIS
LIN {X 114.022,Y 112.488,Z 57.000,A 180.000,B 0.000,C 180.000} C_DIS
LIN {X 111.048,Y 112.488,Z 57.000,A 180.000,B 0.000,C 180.000} C_DIS
LIN {X 111.048,Y 112.488,Z 62.000,A 180.000,B 0.000,C 180.000} C_DIS
LIN {X 97.975,Y 112.488,Z 62.000,A 180.000,B 0.000,C 180.000} C_DIS
LIN {X 97.975,Y 112.488,Z 67.555,A 180.000,B 0.000,C 180.000} C_DIS
LIN {X 97.534,Y 112.488,Z 67.581,A 180.000,B 0.000,C 180.000} C_DIS
LIN {X 97.246,Y 112.488,Z 67.568,A 180.000,B 0.000,C 180.000} C_DIS
LIN {X 97.025,Y 112.488,Z 67.555,A 180.000,B 0.000,C 180.000} C_DIS
LIN {X 97.025,Y 112.488,Z 62.000,A 180.000,B 0.000,C 180.000} C_DIS
LIN {X 64.564,Y 112.488,Z 62.000,A 180.000,B 0.000,C 180.000} C_DIS
LIN {X 64.561,Y 112.488,Z 66.500,A 180.000,B 0.000,C 180.000} C_DIS
LIN {X 64.458,Y 112.488,Z 66.500,A 180.000,B 0.000,C 180.000} C_DIS
LIN {X 64.454,Y 112.488,Z 70.000,A 180.000,B 0.000,C 180.000} C_DIS
LIN {X 52.542,Y 112.488,Z 70.000,A 180.000,B 0.000,C 180.000} C_DIS
LIN {X 52.542,Y 112.488,Z 66.500,A 180.000,B 0.000,C 180.000} C_DIS
LIN {X 52.436,Y 112.488,Z 66.500,A 180.000,B 0.000,C 180.000} C_DIS
LIN {X 52.436,Y 112.488,Z 62.000,A 180.000,B 0.000,C 180.000} C_DIS
LIN {X 43.952,Y 112.488,Z 62.000,A 180.000,B 0.000,C 180.000} C_DIS
LIN {X 43.952,Y 112.488,Z 57.000,A 180.000,B 0.000,C 180.000} C_DIS
LIN {X 40.978,Y 112.488,Z 57.000,A 180.000,B 0.000,C 180.000} C_DIS
LIN {X 40.978,Y 112.488,Z 52.000,A 180.000,B 0.000,C 180.000} C_DIS
LIN {X 32.022,Y 112.488,Z 52.000,A 180.000,B 0.000,C 180.000} C_DIS
LIN {X 32.022,Y 112.488,Z 57.000,A 180.000,B 0.000,C 180.000} C_DIS
LIN {X 11.166,Y 112.488,Z 57.000,A 180.000,B 0.000,C 180.000} C_DIS
LIN {X 11.162,Y 112.488,Z 52.000,A 180.000,B 0.000,C 180.000} C_DIS
LIN {X 2.500,Y 112.488,Z 52.000,A 180.000,B 0.000,C 180.000} C_DIS
LIN {X 2.500,Y 112.488,Z 45.000,A 180.000,B 0.000,C 180.000} C_DIS
LIN {X -0.010,Y 112.488,Z 45.000,A 180.000,B 0.000,C 180.000} C_DIS
; Link Move Starts
LIN {X -0.120,Y 112.488,Z 45.026,A 180.000,B 0.000,C 180.000} C_DIS
LIN {X -0.230,Y 112.488,Z 45.051,A 180.000,B 0.000,C 180.000} C_DIS
LIN {X -0.771,Y 112.800,Z 45.051,A 180.000,B 0.000,C 180.000} C_DIS
LIN {X -0.771,Y 113.425,Z 45.051,A 180.000,B 0.000,C 180.000} C_DIS
LIN {X -0.230,Y 113.738,Z 45.051,A 180.000,B 0.000,C 180.000} C_DIS
LIN {X -0.120,Y 113.738,Z 45.026,A 180.000,B 0.000,C 180.000} C_DIS
LIN {X -0.010,Y 113.738,Z 45.000,A 180.000,B 0.000,C 180.000} C_DIS
; Cutting Move Starts
LIN {X 2.500,Y 113.738,Z 45.000,A 180.000,B 0.000,C 180.000} C_DIS
LIN {X 2.500,Y 113.738,Z 52.000,A 180.000,B 0.000,C 180.000} C_DIS
LIN {X 11.841,Y 113.738,Z 52.000,A 180.000,B 0.000,C 180.000} C_DIS
LIN {X 11.841,Y 113.738,Z 57.000,A 180.000,B 0.000,C 180.000} C_DIS
LIN {X 30.709,Y 113.738,Z 57.000,A 180.000,B 0.000,C 180.000} C_DIS
LIN {X 30.709,Y 113.738,Z 52.000,A 180.000,B 0.000,C 180.000} C_DIS
LIN {X 42.291,Y 113.738,Z 52.000,A 180.000,B 0.000,C 180.000} C_DIS
LIN {X 42.291,Y 113.738,Z 57.000,A 180.000,B 0.000,C 180.000} C_DIS
LIN {X 45.202,Y 113.738,Z 57.000,A 180.000,B 0.000,C 180.000} C_DIS
LIN {X 45.202,Y 113.738,Z 62.000,A 180.000,B 0.000,C 180.000} C_DIS
LIN {X 55.739,Y 113.738,Z 62.000,A 180.000,B 0.000,C 180.000} C_DIS
LIN {X 55.739,Y 113.738,Z 66.500,A 180.000,B 0.000,C 180.000} C_DIS
LIN {X 55.966,Y 113.738,Z 66.500,A 180.000,B 0.000,C 180.000} C_DIS
LIN {X 55.969,Y 113.738,Z 70.000,A 180.000,B 0.000,C 180.000} C_DIS
LIN {X 61.029,Y 113.738,Z 70.000,A 180.000,B 0.000,C 180.000} C_DIS
LIN {X 61.032,Y 113.738,Z 66.500,A 180.000,B 0.000,C 180.000} C_DIS
LIN {X 61.261,Y 113.738,Z 66.500,A 180.000,B 0.000,C 180.000} C_DIS
LIN {X 61.261,Y 113.738,Z 62.000,A 180.000,B 0.000,C 180.000} C_DIS
LIN {X 109.798,Y 113.738,Z 62.000,A 180.000,B 0.000,C 180.000} C_DIS
LIN {X 109.798,Y 113.738,Z 57.000,A 180.000,B 0.000,C 180.000} C_DIS
LIN {X 112.706,Y 113.738,Z 57.000,A 180.000,B 0.000,C 180.000} C_DIS
LIN {X 112.709,Y 113.738,Z 52.000,A 180.000,B 0.000,C 180.000} C_DIS
LIN {X 124.291,Y 113.738,Z 52.000,A 180.000,B 0.000,C 180.000} C_DIS
LIN {X 124.291,Y 113.738,Z 57.000,A 180.000,B 0.000,C 180.000} C_DIS
LIN {X 143.159,Y 113.738,Z 57.000,A 180.000,B 0.000,C 180.000} C_DIS
LIN {X 143.159,Y 113.738,Z 52.000,A 180.000,B 0.000,C 180.000} C_DIS
LIN {X 152.500,Y 113.738,Z 52.000,A 180.000,B 0.000,C 180.000} C_DIS
LIN {X 152.500,Y 113.738,Z 45.000,A 180.000,B 0.000,C 180.000} C_DIS
LIN {X 155.010,Y 113.738,Z 45.000,A 180.000,B 0.000,C 180.000} C_DIS
; Link Move Starts
LIN {X 155.120,Y 113.738,Z 45.026,A 180.000,B 0.000,C 180.000} C_DIS
LIN {X 155.230,Y 113.738,Z 45.051,A 180.000,B 0.000,C 180.000} C_DIS
LIN {X 155.771,Y 114.050,Z 45.051,A 180.000,B 0.000,C 180.000} C_DIS
LIN {X 155.771,Y 114.675,Z 45.051,A 180.000,B 0.000,C 180.000} C_DIS
LIN {X 155.230,Y 114.987,Z 45.051,A 180.000,B 0.000,C 180.000} C_DIS
LIN {X 155.120,Y 114.987,Z 45.026,A 180.000,B 0.000,C 180.000} C_DIS
LIN {X 155.010,Y 114.987,Z 45.000,A 180.000,B 0.000,C 180.000} C_DIS
; Cutting Move Starts
LIN {X 152.500,Y 114.987,Z 45.000,A 180.000,B 0.000,C 180.000} C_DIS
LIN {X 152.500,Y 114.987,Z 52.000,A 180.000,B 0.000,C 180.000} C_DIS
LIN {X 142.454,Y 114.987,Z 52.000,A 180.000,B 0.000,C 180.000} C_DIS
LIN {X 142.454,Y 114.987,Z 57.000,A 180.000,B 0.000,C 180.000} C_DIS
LIN {X 125.122,Y 114.987,Z 57.000,A 180.000,B 0.000,C 180.000} C_DIS
LIN {X 125.122,Y 114.987,Z 52.000,A 180.000,B 0.000,C 180.000} C_DIS
LIN {X 111.878,Y 114.987,Z 52.000,A 180.000,B 0.000,C 180.000} C_DIS
LIN {X 111.878,Y 114.987,Z 57.000,A 180.000,B 0.000,C 180.000} C_DIS
LIN {X 108.548,Y 114.987,Z 57.000,A 180.000,B 0.000,C 180.000} C_DIS
LIN {X 108.548,Y 114.987,Z 62.000,A 180.000,B 0.000,C 180.000} C_DIS
LIN {X 46.452,Y 114.987,Z 62.000,A 180.000,B 0.000,C 180.000} C_DIS
LIN {X 46.452,Y 114.987,Z 57.000,A 180.000,B 0.000,C 180.000} C_DIS
LIN {X 43.122,Y 114.987,Z 57.000,A 180.000,B 0.000,C 180.000} C_DIS
LIN {X 43.122,Y 114.987,Z 52.000,A 180.000,B 0.000,C 180.000} C_DIS
LIN {X 29.878,Y 114.987,Z 52.000,A 180.000,B 0.000,C 180.000} C_DIS
LIN {X 29.878,Y 114.987,Z 57.000,A 180.000,B 0.000,C 180.000} C_DIS
LIN {X 12.546,Y 114.987,Z 57.000,A 180.000,B 0.000,C 180.000} C_DIS
LIN {X 12.546,Y 114.987,Z 52.000,A 180.000,B 0.000,C 180.000} C_DIS
LIN {X 2.500,Y 114.987,Z 52.000,A 180.000,B 0.000,C 180.000} C_DIS
LIN {X 2.500,Y 114.987,Z 45.000,A 180.000,B 0.000,C 180.000} C_DIS
LIN {X -0.010,Y 114.987,Z 45.000,A 180.000,B 0.000,C 180.000} C_DIS
; Link Move Starts
LIN {X -0.120,Y 114.987,Z 45.026,A 180.000,B 0.000,C 180.000} C_DIS
LIN {X -0.230,Y 114.987,Z 45.051,A 180.000,B 0.000,C 180.000} C_DIS
LIN {X -0.771,Y 115.300,Z 45.051,A 180.000,B 0.000,C 180.000} C_DIS
LIN {X -0.771,Y 115.925,Z 45.051,A 180.000,B 0.000,C 180.000} C_DIS
LIN {X -0.230,Y 116.237,Z 45.051,A 180.000,B 0.000,C 180.000} C_DIS
LIN {X -0.120,Y 116.237,Z 45.026,A 180.000,B 0.000,C 180.000} C_DIS
LIN {X -0.010,Y 116.237,Z 45.000,A 180.000,B 0.000,C 180.000} C_DIS
; Cutting Move Starts
LIN {X 2.500,Y 116.237,Z 45.000,A 180.000,B 0.000,C 180.000} C_DIS
LIN {X 2.500,Y 116.237,Z 52.000,A 180.000,B 0.000,C 180.000} C_DIS
LIN {X 13.281,Y 116.237,Z 52.000,A 180.000,B 0.000,C 180.000} C_DIS
LIN {X 13.281,Y 116.237,Z 57.000,A 180.000,B 0.000,C 180.000} C_DIS
LIN {X 29.352,Y 116.237,Z 57.000,A 180.000,B 0.000,C 180.000} C_DIS
LIN {X 29.352,Y 116.237,Z 52.000,A 180.000,B 0.000,C 180.000} C_DIS
LIN {X 43.646,Y 116.237,Z 52.000,A 180.000,B 0.000,C 180.000} C_DIS
LIN {X 43.648,Y 116.237,Z 57.000,A 180.000,B 0.000,C 180.000} C_DIS
LIN {X 47.702,Y 116.237,Z 57.000,A 180.000,B 0.000,C 180.000} C_DIS
LIN {X 47.702,Y 116.237,Z 62.000,A 180.000,B 0.000,C 180.000} C_DIS
LIN {X 107.297,Y 116.237,Z 62.000,A 180.000,B 0.000,C 180.000} C_DIS
LIN {X 107.298,Y 116.237,Z 57.000,A 180.000,B 0.000,C 180.000} C_DIS
LIN {X 111.352,Y 116.237,Z 57.000,A 180.000,B 0.000,C 180.000} C_DIS
LIN {X 111.352,Y 116.237,Z 52.000,A 180.000,B 0.000,C 180.000} C_DIS
LIN {X 125.648,Y 116.237,Z 52.000,A 180.000,B 0.000,C 180.000} C_DIS
LIN {X 125.648,Y 116.237,Z 57.000,A 180.000,B 0.000,C 180.000} C_DIS
LIN {X 141.719,Y 116.237,Z 57.000,A 180.000,B 0.000,C 180.000} C_DIS
LIN {X 141.719,Y 116.237,Z 52.000,A 180.000,B 0.000,C 180.000} C_DIS
LIN {X 152.500,Y 116.237,Z 52.000,A 180.000,B 0.000,C 180.000} C_DIS
LIN {X 152.500,Y 116.237,Z 45.000,A 180.000,B 0.000,C 180.000} C_DIS
LIN {X 155.010,Y 116.237,Z 45.000,A 180.000,B 0.000,C 180.000} C_DIS
; Link Move Starts
LIN {X 155.120,Y 116.237,Z 45.026,A 180.000,B 0.000,C 180.000} C_DIS
LIN {X 155.230,Y 116.237,Z 45.051,A 180.000,B 0.000,C 180.000} C_DIS
LIN {X 155.771,Y 116.550,Z 45.051,A 180.000,B 0.000,C 180.000} C_DIS
LIN {X 155.771,Y 117.175,Z 45.051,A 180.000,B 0.000,C 180.000} C_DIS
LIN {X 155.230,Y 117.487,Z 45.051,A 180.000,B 0.000,C 180.000} C_DIS
LIN {X 155.120,Y 117.487,Z 45.026,A 180.000,B 0.000,C 180.000} C_DIS
LIN {X 155.010,Y 117.487,Z 45.000,A 180.000,B 0.000,C 180.000} C_DIS
; Cutting Move Starts
LIN {X 152.500,Y 117.487,Z 45.000,A 180.000,B 0.000,C 180.000} C_DIS
LIN {X 152.500,Y 117.487,Z 52.000,A 180.000,B 0.000,C 180.000} C_DIS
LIN {X 140.951,Y 117.487,Z 52.000,A 180.000,B 0.000,C 180.000} C_DIS
LIN {X 140.951,Y 117.487,Z 57.000,A 180.000,B 0.000,C 180.000} C_DIS
LIN {X 125.928,Y 117.487,Z 57.000,A 180.000,B 0.000,C 180.000} C_DIS
LIN {X 125.928,Y 117.487,Z 52.000,A 180.000,B 0.000,C 180.000} C_DIS
LIN {X 111.072,Y 117.487,Z 52.000,A 180.000,B 0.000,C 180.000} C_DIS
LIN {X 111.071,Y 117.487,Z 57.000,A 180.000,B 0.000,C 180.000} C_DIS
LIN {X 106.048,Y 117.487,Z 57.000,A 180.000,B 0.000,C 180.000} C_DIS
LIN {X 106.048,Y 117.487,Z 62.000,A 180.000,B 0.000,C 180.000} C_DIS
LIN {X 48.952,Y 117.487,Z 62.000,A 180.000,B 0.000,C 180.000} C_DIS
LIN {X 48.952,Y 117.487,Z 57.000,A 180.000,B 0.000,C 180.000} C_DIS
LIN {X 43.928,Y 117.487,Z 57.000,A 180.000,B 0.000,C 180.000} C_DIS
LIN {X 43.928,Y 117.487,Z 52.000,A 180.000,B 0.000,C 180.000} C_DIS
LIN {X 29.072,Y 117.487,Z 52.000,A 180.000,B 0.000,C 180.000} C_DIS
LIN {X 29.067,Y 117.487,Z 57.000,A 180.000,B 0.000,C 180.000} C_DIS
LIN {X 14.049,Y 117.487,Z 57.000,A 180.000,B 0.000,C 180.000} C_DIS
LIN {X 14.049,Y 117.487,Z 52.000,A 180.000,B 0.000,C 180.000} C_DIS
LIN {X 2.500,Y 117.487,Z 52.000,A 180.000,B 0.000,C 180.000} C_DIS
LIN {X 2.500,Y 117.487,Z 45.000,A 180.000,B 0.000,C 180.000} C_DIS
LIN {X -0.010,Y 117.487,Z 45.000,A 180.000,B 0.000,C 180.000} C_DIS
; Link Move Starts
LIN {X -0.120,Y 117.487,Z 45.026,A 180.000,B 0.000,C 180.000} C_DIS
LIN {X -0.230,Y 117.487,Z 45.051,A 180.000,B 0.000,C 180.000} C_DIS
LIN {X -0.771,Y 117.800,Z 45.051,A 180.000,B 0.000,C 180.000} C_DIS
LIN {X -0.771,Y 118.425,Z 45.051,A 180.000,B 0.000,C 180.000} C_DIS
LIN {X -0.230,Y 118.737,Z 45.051,A 180.000,B 0.000,C 180.000} C_DIS
LIN {X -0.120,Y 118.737,Z 45.026,A 180.000,B 0.000,C 180.000} C_DIS
LIN {X -0.010,Y 118.737,Z 45.000,A 180.000,B 0.000,C 180.000} C_DIS
; Cutting Move Starts
LIN {X 2.500,Y 118.737,Z 45.000,A 180.000,B 0.000,C 180.000} C_DIS
LIN {X 2.500,Y 118.737,Z 52.000,A 180.000,B 0.000,C 180.000} C_DIS
LIN {X 14.857,Y 118.737,Z 52.000,A 180.000,B 0.000,C 180.000} C_DIS
LIN {X 14.857,Y 118.737,Z 57.000,A 180.000,B 0.000,C 180.000} C_DIS
LIN {X 29.008,Y 118.737,Z 57.000,A 180.000,B 0.000,C 180.000} C_DIS
LIN {X 29.009,Y 118.737,Z 52.000,A 180.000,B 0.000,C 180.000} C_DIS
LIN {X 43.988,Y 118.737,Z 52.000,A 180.000,B 0.000,C 180.000} C_DIS
LIN {X 43.991,Y 118.737,Z 57.000,A 180.000,B 0.000,C 180.000} C_DIS
LIN {X 50.202,Y 118.737,Z 57.000,A 180.000,B 0.000,C 180.000} C_DIS
LIN {X 50.202,Y 118.737,Z 62.000,A 180.000,B 0.000,C 180.000} C_DIS
LIN {X 104.795,Y 118.737,Z 62.000,A 180.000,B 0.000,C 180.000} C_DIS
LIN {X 104.798,Y 118.737,Z 57.000,A 180.000,B 0.000,C 180.000} C_DIS
LIN {X 111.008,Y 118.737,Z 57.000,A 180.000,B 0.000,C 180.000} C_DIS
LIN {X 111.009,Y 118.737,Z 52.000,A 180.000,B 0.000,C 180.000} C_DIS
LIN {X 125.991,Y 118.737,Z 52.000,A 180.000,B 0.000,C 180.000} C_DIS
LIN {X 125.991,Y 118.737,Z 57.000,A 180.000,B 0.000,C 180.000} C_DIS
LIN {X 140.143,Y 118.737,Z 57.000,A 180.000,B 0.000,C 180.000} C_DIS
LIN {X 140.143,Y 118.737,Z 52.000,A 180.000,B 0.000,C 180.000} C_DIS
LIN {X 152.500,Y 118.737,Z 52.000,A 180.000,B 0.000,C 180.000} C_DIS
LIN {X 152.500,Y 118.737,Z 45.000,A 180.000,B 0.000,C 180.000} C_DIS
LIN {X 155.010,Y 118.737,Z 45.000,A 180.000,B 0.000,C 180.000} C_DIS
; Link Move Starts
LIN {X 155.120,Y 118.737,Z 45.026,A 180.000,B 0.000,C 180.000} C_DIS
LIN {X 155.230,Y 118.737,Z 45.051,A 180.000,B 0.000,C 180.000} C_DIS
LIN {X 155.771,Y 119.050,Z 45.051,A 180.000,B 0.000,C 180.000} C_DIS
LIN {X 155.771,Y 119.675,Z 45.051,A 180.000,B 0.000,C 180.000} C_DIS
LIN {X 155.230,Y 119.987,Z 45.051,A 180.000,B 0.000,C 180.000} C_DIS
LIN {X 155.120,Y 119.987,Z 45.026,A 180.000,B 0.000,C 180.000} C_DIS
LIN {X 155.010,Y 119.987,Z 45.000,A 180.000,B 0.000,C 180.000} C_DIS
; Cutting Move Starts
LIN {X 152.500,Y 119.987,Z 45.000,A 180.000,B 0.000,C 180.000} C_DIS
LIN {X 152.500,Y 119.987,Z 52.000,A 180.000,B 0.000,C 180.000} C_DIS
LIN {X 139.300,Y 119.987,Z 52.000,A 180.000,B 0.000,C 180.000} C_DIS
LIN {X 139.300,Y 119.987,Z 57.000,A 180.000,B 0.000,C 180.000} C_DIS
LIN {X 125.848,Y 119.987,Z 57.000,A 180.000,B 0.000,C 180.000} C_DIS
LIN {X 125.847,Y 119.987,Z 52.000,A 180.000,B 0.000,C 180.000} C_DIS
LIN {X 111.152,Y 119.987,Z 52.000,A 180.000,B 0.000,C 180.000} C_DIS
LIN {X 111.152,Y 119.987,Z 57.000,A 180.000,B 0.000,C 180.000} C_DIS
LIN {X 103.548,Y 119.987,Z 57.000,A 180.000,B 0.000,C 180.000} C_DIS
LIN {X 103.546,Y 119.987,Z 62.000,A 180.000,B 0.000,C 180.000} C_DIS
LIN {X 51.452,Y 119.987,Z 62.000,A 180.000,B 0.000,C 180.000} C_DIS
LIN {X 51.451,Y 119.987,Z 57.000,A 180.000,B 0.000,C 180.000} C_DIS
LIN {X 43.848,Y 119.987,Z 57.000,A 180.000,B 0.000,C 180.000} C_DIS
LIN {X 43.848,Y 119.987,Z 52.000,A 180.000,B 0.000,C 180.000} C_DIS
LIN {X 29.152,Y 119.987,Z 52.000,A 180.000,B 0.000,C 180.000} C_DIS
LIN {X 29.152,Y 119.987,Z 57.000,A 180.000,B 0.000,C 180.000} C_DIS
LIN {X 15.700,Y 119.987,Z 57.000,A 180.000,B 0.000,C 180.000} C_DIS
LIN {X 15.700,Y 119.987,Z 52.000,A 180.000,B 0.000,C 180.000} C_DIS
LIN {X 2.500,Y 119.987,Z 52.000,A 180.000,B 0.000,C 180.000} C_DIS
LIN {X 2.500,Y 119.987,Z 45.000,A 180.000,B 0.000,C 180.000} C_DIS
LIN {X -0.010,Y 119.987,Z 45.000,A 180.000,B 0.000,C 180.000} C_DIS
; Link Move Starts
LIN {X -0.120,Y 119.987,Z 45.026,A 180.000,B 0.000,C 180.000} C_DIS
LIN {X -0.230,Y 119.987,Z 45.051,A 180.000,B 0.000,C 180.000} C_DIS
LIN {X -0.771,Y 120.300,Z 45.051,A 180.000,B 0.000,C 180.000} C_DIS
LIN {X -0.771,Y 120.924,Z 45.051,A 180.000,B 0.000,C 180.000} C_DIS
LIN {X -0.230,Y 121.237,Z 45.051,A 180.000,B 0.000,C 180.000} C_DIS
LIN {X -0.120,Y 121.237,Z 45.026,A 180.000,B 0.000,C 180.000} C_DIS
LIN {X -0.010,Y 121.237,Z 45.000,A 180.000,B 0.000,C 180.000} C_DIS
; Cutting Move Starts
LIN {X 2.497,Y 121.237,Z 45.000,A 180.000,B 0.000,C 180.000} C_DIS
LIN {X 2.500,Y 121.237,Z 52.000,A 180.000,B 0.000,C 180.000} C_DIS
LIN {X 16.579,Y 121.237,Z 52.000,A 180.000,B 0.000,C 180.000} C_DIS
LIN {X 16.579,Y 121.237,Z 57.000,A 180.000,B 0.000,C 180.000} C_DIS
LIN {X 29.519,Y 121.237,Z 57.000,A 180.000,B 0.000,C 180.000} C_DIS
LIN {X 29.519,Y 121.237,Z 52.000,A 180.000,B 0.000,C 180.000} C_DIS
LIN {X 43.481,Y 121.237,Z 52.000,A 180.000,B 0.000,C 180.000} C_DIS
LIN {X 43.481,Y 121.237,Z 57.000,A 180.000,B 0.000,C 180.000} C_DIS
LIN {X 52.701,Y 121.237,Z 57.000,A 180.000,B 0.000,C 180.000} C_DIS
LIN {X 52.701,Y 121.237,Z 62.000,A 180.000,B 0.000,C 180.000} C_DIS
LIN {X 102.299,Y 121.237,Z 62.000,A 180.000,B 0.000,C 180.000} C_DIS
LIN {X 102.299,Y 121.237,Z 57.000,A 180.000,B 0.000,C 180.000} C_DIS
LIN {X 111.519,Y 121.237,Z 57.000,A 180.000,B 0.000,C 180.000} C_DIS
LIN {X 111.519,Y 121.237,Z 52.000,A 180.000,B 0.000,C 180.000} C_DIS
LIN {X 125.481,Y 121.237,Z 52.000,A 180.000,B 0.000,C 180.000} C_DIS
LIN {X 125.481,Y 121.237,Z 57.000,A 180.000,B 0.000,C 180.000} C_DIS
LIN {X 138.420,Y 121.237,Z 57.000,A 180.000,B 0.000,C 180.000} C_DIS
LIN {X 138.421,Y 121.237,Z 52.000,A 180.000,B 0.000,C 180.000} C_DIS
LIN {X 152.500,Y 121.237,Z 52.000,A 180.000,B 0.000,C 180.000} C_DIS
LIN {X 152.500,Y 121.237,Z 45.000,A 180.000,B 0.000,C 180.000} C_DIS
LIN {X 155.010,Y 121.237,Z 45.000,A 180.000,B 0.000,C 180.000} C_DIS
; Link Move Starts
LIN {X 155.120,Y 121.237,Z 45.026,A 180.000,B 0.000,C 180.000} C_DIS
LIN {X 155.230,Y 121.237,Z 45.051,A 180.000,B 0.000,C 180.000} C_DIS
LIN {X 155.771,Y 121.549,Z 45.051,A 180.000,B 0.000,C 180.000} C_DIS
LIN {X 155.771,Y 122.174,Z 45.051,A 180.000,B 0.000,C 180.000} C_DIS
LIN {X 155.230,Y 122.487,Z 45.051,A 180.000,B 0.000,C 180.000} C_DIS
LIN {X 155.120,Y 122.487,Z 45.026,A 180.000,B 0.000,C 180.000} C_DIS
LIN {X 155.010,Y 122.487,Z 45.000,A 180.000,B 0.000,C 180.000} C_DIS
; Cutting Move Starts
LIN {X 152.500,Y 122.487,Z 45.000,A 180.000,B 0.000,C 180.000} C_DIS
LIN {X 152.500,Y 122.487,Z 52.000,A 180.000,B 0.000,C 180.000} C_DIS
LIN {X 137.504,Y 122.487,Z 52.000,A 180.000,B 0.000,C 180.000} C_DIS
LIN {X 137.501,Y 122.487,Z 57.000,A 180.000,B 0.000,C 180.000} C_DIS
LIN {X 124.850,Y 122.487,Z 57.000,A 180.000,B 0.000,C 180.000} C_DIS
LIN {X 124.847,Y 122.487,Z 52.000,A 180.000,B 0.000,C 180.000} C_DIS
LIN {X 112.150,Y 122.487,Z 52.000,A 180.000,B 0.000,C 180.000} C_DIS
LIN {X 112.147,Y 122.487,Z 57.000,A 180.000,B 0.000,C 180.000} C_DIS
LIN {X 101.049,Y 122.487,Z 57.000,A 180.000,B 0.000,C 180.000} C_DIS
LIN {X 101.049,Y 122.487,Z 62.000,A 180.000,B 0.000,C 180.000} C_DIS
LIN {X 53.951,Y 122.487,Z 62.000,A 180.000,B 0.000,C 180.000} C_DIS
LIN {X 53.951,Y 122.487,Z 57.000,A 180.000,B 0.000,C 180.000} C_DIS
LIN {X 42.850,Y 122.487,Z 57.000,A 180.000,B 0.000,C 180.000} C_DIS
LIN {X 42.850,Y 122.487,Z 52.000,A 180.000,B 0.000,C 180.000} C_DIS
LIN {X 30.150,Y 122.487,Z 52.000,A 180.000,B 0.000,C 180.000} C_DIS
LIN {X 30.150,Y 122.487,Z 57.000,A 180.000,B 0.000,C 180.000} C_DIS
LIN {X 17.496,Y 122.487,Z 57.000,A 180.000,B 0.000,C 180.000} C_DIS
LIN {X 17.496,Y 122.487,Z 52.000,A 180.000,B 0.000,C 180.000} C_DIS
LIN {X 2.500,Y 122.487,Z 52.000,A 180.000,B 0.000,C 180.000} C_DIS
LIN {X 2.496,Y 122.487,Z 45.000,A 180.000,B 0.000,C 180.000} C_DIS
LIN {X -0.010,Y 122.487,Z 45.000,A 180.000,B 0.000,C 180.000} C_DIS
; Link Move Starts
LIN {X -0.120,Y 122.487,Z 45.026,A 180.000,B 0.000,C 180.000} C_DIS
LIN {X -0.230,Y 122.487,Z 45.051,A 180.000,B 0.000,C 180.000} C_DIS
LIN {X -0.771,Y 122.799,Z 45.051,A 180.000,B 0.000,C 180.000} C_DIS
LIN {X -0.771,Y 123.424,Z 45.051,A 180.000,B 0.000,C 180.000} C_DIS
LIN {X -0.230,Y 123.737,Z 45.051,A 180.000,B 0.000,C 180.000} C_DIS
LIN {X -0.120,Y 123.737,Z 45.026,A 180.000,B 0.000,C 180.000} C_DIS
LIN {X -0.010,Y 123.737,Z 45.000,A 180.000,B 0.000,C 180.000} C_DIS
; Cutting Move Starts
LIN {X 2.500,Y 123.737,Z 45.000,A 180.000,B 0.000,C 180.000} C_DIS
LIN {X 2.500,Y 123.737,Z 52.000,A 180.000,B 0.000,C 180.000} C_DIS
LIN {X 18.453,Y 123.737,Z 52.000,A 180.000,B 0.000,C 180.000} C_DIS
LIN {X 18.453,Y 123.737,Z 57.000,A 180.000,B 0.000,C 180.000} C_DIS
LIN {X 31.134,Y 123.737,Z 57.000,A 180.000,B 0.000,C 180.000} C_DIS
LIN {X 31.137,Y 123.737,Z 52.000,A 180.000,B 0.000,C 180.000} C_DIS
LIN {X 41.863,Y 123.737,Z 52.000,A 180.000,B 0.000,C 180.000} C_DIS
LIN {X 41.863,Y 123.737,Z 57.000,A 180.000,B 0.000,C 180.000} C_DIS
LIN {X 55.201,Y 123.737,Z 57.000,A 180.000,B 0.000,C 180.000} C_DIS
LIN {X 55.201,Y 123.737,Z 62.000,A 180.000,B 0.000,C 180.000} C_DIS
LIN {X 99.799,Y 123.737,Z 62.000,A 180.000,B 0.000,C 180.000} C_DIS
LIN {X 99.799,Y 123.737,Z 57.000,A 180.000,B 0.000,C 180.000} C_DIS
LIN {X 113.134,Y 123.737,Z 57.000,A 180.000,B 0.000,C 180.000} C_DIS
LIN {X 113.137,Y 123.737,Z 52.000,A 180.000,B 0.000,C 180.000} C_DIS
LIN {X 123.859,Y 123.737,Z 52.000,A 180.000,B 0.000,C 180.000} C_DIS
LIN {X 123.863,Y 123.737,Z 57.000,A 180.000,B 0.000,C 180.000} C_DIS
LIN {X 136.547,Y 123.737,Z 57.000,A 180.000,B 0.000,C 180.000} C_DIS
LIN {X 136.547,Y 123.737,Z 52.000,A 180.000,B 0.000,C 180.000} C_DIS
LIN {X 152.500,Y 123.737,Z 52.000,A 180.000,B 0.000,C 180.000} C_DIS
LIN {X 152.500,Y 123.737,Z 45.000,A 180.000,B 0.000,C 180.000} C_DIS
LIN {X 155.010,Y 123.737,Z 45.000,A 180.000,B 0.000,C 180.000} C_DIS
; Link Move Starts
LIN {X 155.120,Y 123.737,Z 45.026,A 180.000,B 0.000,C 180.000} C_DIS
LIN {X 155.230,Y 123.737,Z 45.051,A 180.000,B 0.000,C 180.000} C_DIS
LIN {X 155.771,Y 124.049,Z 45.051,A 180.000,B 0.000,C 180.000} C_DIS
LIN {X 155.771,Y 124.674,Z 45.051,A 180.000,B 0.000,C 180.000} C_DIS
LIN {X 155.230,Y 124.987,Z 45.051,A 180.000,B 0.000,C 180.000} C_DIS
LIN {X 155.120,Y 124.987,Z 45.026,A 180.000,B 0.000,C 180.000} C_DIS
LIN {X 155.010,Y 124.987,Z 45.000,A 180.000,B 0.000,C 180.000} C_DIS
; Cutting Move Starts
LIN {X 152.500,Y 124.987,Z 45.000,A 180.000,B 0.000,C 180.000} C_DIS
LIN {X 152.500,Y 124.987,Z 52.000,A 180.000,B 0.000,C 180.000} C_DIS
LIN {X 135.547,Y 124.987,Z 52.000,A 180.000,B 0.000,C 180.000} C_DIS
LIN {X 135.542,Y 124.987,Z 57.000,A 180.000,B 0.000,C 180.000} C_DIS
LIN {X 122.256,Y 124.987,Z 57.000,A 180.000,B 0.000,C 180.000} C_DIS
LIN {X 122.256,Y 124.987,Z 52.000,A 180.000,B 0.000,C 180.000} C_DIS
LIN {X 114.744,Y 124.987,Z 52.000,A 180.000,B 0.000,C 180.000} C_DIS
LIN {X 114.741,Y 124.987,Z 57.000,A 180.000,B 0.000,C 180.000} C_DIS
LIN {X 98.549,Y 124.987,Z 57.000,A 180.000,B 0.000,C 180.000} C_DIS
LIN {X 98.549,Y 124.987,Z 62.000,A 180.000,B 0.000,C 180.000} C_DIS
LIN {X 56.451,Y 124.987,Z 62.000,A 180.000,B 0.000,C 180.000} C_DIS
LIN {X 56.451,Y 124.987,Z 57.000,A 180.000,B 0.000,C 180.000} C_DIS
LIN {X 40.256,Y 124.987,Z 57.000,A 180.000,B 0.000,C 180.000} C_DIS
LIN {X 40.256,Y 124.987,Z 52.000,A 180.000,B 0.000,C 180.000} C_DIS
LIN {X 32.744,Y 124.987,Z 52.000,A 180.000,B 0.000,C 180.000} C_DIS
LIN {X 32.741,Y 124.987,Z 57.000,A 180.000,B 0.000,C 180.000} C_DIS
LIN {X 19.453,Y 124.987,Z 57.000,A 180.000,B 0.000,C 180.000} C_DIS
LIN {X 19.453,Y 124.987,Z 52.000,A 180.000,B 0.000,C 180.000} C_DIS
LIN {X 2.500,Y 124.987,Z 52.000,A 180.000,B 0.000,C 180.000} C_DIS
LIN {X 2.495,Y 124.987,Z 45.000,A 180.000,B 0.000,C 180.000} C_DIS
LIN {X -0.010,Y 124.987,Z 45.000,A 180.000,B 0.000,C 180.000} C_DIS
; Link Move Starts
LIN {X -0.120,Y 124.987,Z 45.026,A 180.000,B 0.000,C 180.000} C_DIS
LIN {X -0.230,Y 124.987,Z 45.051,A 180.000,B 0.000,C 180.000} C_DIS
LIN {X -0.771,Y 125.299,Z 45.051,A 180.000,B 0.000,C 180.000} C_DIS
LIN {X -0.771,Y 125.924,Z 45.051,A 180.000,B 0.000,C 180.000} C_DIS
LIN {X -0.230,Y 126.237,Z 45.051,A 180.000,B 0.000,C 180.000} C_DIS
LIN {X -0.120,Y 126.237,Z 45.026,A 180.000,B 0.000,C 180.000} C_DIS
LIN {X -0.010,Y 126.237,Z 45.000,A 180.000,B 0.000,C 180.000} C_DIS
; Cutting Move Starts
LIN {X 2.499,Y 126.237,Z 45.000,A 180.000,B 0.000,C 180.000} C_DIS
LIN {X 2.500,Y 126.237,Z 52.000,A 180.000,B 0.000,C 180.000} C_DIS
LIN {X 20.495,Y 126.237,Z 52.000,A 180.000,B 0.000,C 180.000} C_DIS
LIN {X 20.497,Y 126.237,Z 57.000,A 180.000,B 0.000,C 180.000} C_DIS
LIN {X 57.701,Y 126.237,Z 57.000,A 180.000,B 0.000,C 180.000} C_DIS
LIN {X 57.701,Y 126.237,Z 62.000,A 180.000,B 0.000,C 180.000} C_DIS
LIN {X 97.297,Y 126.237,Z 62.000,A 180.000,B 0.000,C 180.000} C_DIS
LIN {X 97.299,Y 126.237,Z 57.000,A 180.000,B 0.000,C 180.000} C_DIS
LIN {X 134.502,Y 126.237,Z 57.000,A 180.000,B 0.000,C 180.000} C_DIS
LIN {X 134.503,Y 126.237,Z 52.000,A 180.000,B 0.000,C 180.000} C_DIS
LIN {X 152.500,Y 126.237,Z 52.000,A 180.000,B 0.000,C 180.000} C_DIS
LIN {X 152.500,Y 126.237,Z 45.000,A 180.000,B 0.000,C 180.000} C_DIS
LIN {X 155.010,Y 126.237,Z 45.000,A 180.000,B 0.000,C 180.000} C_DIS
; Link Move Starts
LIN {X 155.120,Y 126.237,Z 45.026,A 180.000,B 0.000,C 180.000} C_DIS
LIN {X 155.230,Y 126.237,Z 45.051,A 180.000,B 0.000,C 180.000} C_DIS
LIN {X 155.771,Y 126.549,Z 45.051,A 180.000,B 0.000,C 180.000} C_DIS
LIN {X 155.771,Y 127.174,Z 45.051,A 180.000,B 0.000,C 180.000} C_DIS
LIN {X 155.230,Y 127.486,Z 45.051,A 180.000,B 0.000,C 180.000} C_DIS
LIN {X 155.120,Y 127.486,Z 45.026,A 180.000,B 0.000,C 180.000} C_DIS
LIN {X 155.010,Y 127.486,Z 45.000,A 180.000,B 0.000,C 180.000} C_DIS
; Cutting Move Starts
LIN {X 152.500,Y 127.486,Z 45.000,A 180.000,B 0.000,C 180.000} C_DIS
LIN {X 152.500,Y 127.486,Z 52.000,A 180.000,B 0.000,C 180.000} C_DIS
LIN {X 133.411,Y 127.486,Z 52.000,A 180.000,B 0.000,C 180.000} C_DIS
LIN {X 133.411,Y 127.486,Z 57.000,A 180.000,B 0.000,C 180.000} C_DIS
LIN {X 96.049,Y 127.486,Z 57.000,A 180.000,B 0.000,C 180.000} C_DIS
LIN {X 96.049,Y 127.486,Z 62.000,A 180.000,B 0.000,C 180.000} C_DIS
LIN {X 58.951,Y 127.486,Z 62.000,A 180.000,B 0.000,C 180.000} C_DIS
LIN {X 58.950,Y 127.486,Z 57.000,A 180.000,B 0.000,C 180.000} C_DIS
LIN {X 21.589,Y 127.486,Z 57.000,A 180.000,B 0.000,C 180.000} C_DIS
LIN {X 21.589,Y 127.486,Z 52.000,A 180.000,B 0.000,C 180.000} C_DIS
LIN {X 2.500,Y 127.486,Z 52.000,A 180.000,B 0.000,C 180.000} C_DIS
LIN {X 2.500,Y 127.486,Z 45.000,A 180.000,B 0.000,C 180.000} C_DIS
LIN {X -0.010,Y 127.486,Z 45.000,A 180.000,B 0.000,C 180.000} C_DIS
; Link Move Starts
LIN {X -0.120,Y 127.486,Z 45.026,A 180.000,B 0.000,C 180.000} C_DIS
LIN {X -0.230,Y 127.486,Z 45.051,A 180.000,B 0.000,C 180.000} C_DIS
LIN {X -0.771,Y 127.799,Z 45.051,A 180.000,B 0.000,C 180.000} C_DIS
LIN {X -0.771,Y 128.424,Z 45.051,A 180.000,B 0.000,C 180.000} C_DIS
LIN {X -0.230,Y 128.736,Z 45.051,A 180.000,B 0.000,C 180.000} C_DIS
LIN {X -0.120,Y 128.736,Z 45.026,A 180.000,B 0.000,C 180.000} C_DIS
LIN {X -0.010,Y 128.736,Z 45.000,A 180.000,B 0.000,C 180.000} C_DIS
; Cutting Move Starts
LIN {X 2.498,Y 128.736,Z 45.000,A 180.000,B 0.000,C 180.000} C_DIS
LIN {X 2.500,Y 128.736,Z 52.000,A 180.000,B 0.000,C 180.000} C_DIS
LIN {X 22.731,Y 128.736,Z 52.000,A 180.000,B 0.000,C 180.000} C_DIS
LIN {X 22.731,Y 128.736,Z 57.000,A 180.000,B 0.000,C 180.000} C_DIS
LIN {X 60.201,Y 128.736,Z 57.000,A 180.000,B 0.000,C 180.000} C_DIS
LIN {X 60.201,Y 128.736,Z 62.000,A 180.000,B 0.000,C 180.000} C_DIS
LIN {X 94.799,Y 128.736,Z 62.000,A 180.000,B 0.000,C 180.000} C_DIS
LIN {X 94.799,Y 128.736,Z 57.000,A 180.000,B 0.000,C 180.000} C_DIS
LIN {X 132.267,Y 128.736,Z 57.000,A 180.000,B 0.000,C 180.000} C_DIS
LIN {X 132.269,Y 128.736,Z 52.000,A 180.000,B 0.000,C 180.000} C_DIS
LIN {X 152.500,Y 128.736,Z 52.000,A 180.000,B 0.000,C 180.000} C_DIS
LIN {X 152.500,Y 128.736,Z 45.000,A 180.000,B 0.000,C 180.000} C_DIS
LIN {X 155.010,Y 128.736,Z 45.000,A 180.000,B 0.000,C 180.000} C_DIS
; Link Move Starts
LIN {X 155.120,Y 128.736,Z 45.026,A 180.000,B 0.000,C 180.000} C_DIS
LIN {X 155.230,Y 128.736,Z 45.051,A 180.000,B 0.000,C 180.000} C_DIS
LIN {X 155.771,Y 129.049,Z 45.051,A 180.000,B 0.000,C 180.000} C_DIS
LIN {X 155.771,Y 129.674,Z 45.051,A 180.000,B 0.000,C 180.000} C_DIS
LIN {X 155.230,Y 129.986,Z 45.051,A 180.000,B 0.000,C 180.000} C_DIS
LIN {X 155.120,Y 129.986,Z 45.026,A 180.000,B 0.000,C 180.000} C_DIS
LIN {X 155.010,Y 129.986,Z 45.000,A 180.000,B 0.000,C 180.000} C_DIS
; Cutting Move Starts
LIN {X 152.500,Y 129.986,Z 45.000,A 180.000,B 0.000,C 180.000} C_DIS
LIN {X 152.500,Y 129.986,Z 52.000,A 180.000,B 0.000,C 180.000} C_DIS
LIN {X 131.073,Y 129.986,Z 52.000,A 180.000,B 0.000,C 180.000} C_DIS
LIN {X 131.073,Y 129.986,Z 57.000,A 180.000,B 0.000,C 180.000} C_DIS
LIN {X 93.549,Y 129.986,Z 57.000,A 180.000,B 0.000,C 180.000} C_DIS
LIN {X 93.546,Y 129.986,Z 62.000,A 180.000,B 0.000,C 180.000} C_DIS
LIN {X 61.451,Y 129.986,Z 62.000,A 180.000,B 0.000,C 180.000} C_DIS
LIN {X 61.451,Y 129.986,Z 57.000,A 180.000,B 0.000,C 180.000} C_DIS
LIN {X 23.927,Y 129.986,Z 57.000,A 180.000,B 0.000,C 180.000} C_DIS
LIN {X 23.924,Y 129.986,Z 52.000,A 180.000,B 0.000,C 180.000} C_DIS
LIN {X 2.500,Y 129.986,Z 52.000,A 180.000,B 0.000,C 180.000} C_DIS
LIN {X 2.500,Y 129.986,Z 45.000,A 180.000,B 0.000,C 180.000} C_DIS
LIN {X -0.010,Y 129.986,Z 45.000,A 180.000,B 0.000,C 180.000} C_DIS
; Link Move Starts
LIN {X -0.120,Y 129.986,Z 45.026,A 180.000,B 0.000,C 180.000} C_DIS
LIN {X -0.230,Y 129.986,Z 45.051,A 180.000,B 0.000,C 180.000} C_DIS
LIN {X -0.771,Y 130.299,Z 45.051,A 180.000,B 0.000,C 180.000} C_DIS
LIN {X -0.771,Y 130.924,Z 45.051,A 180.000,B 0.000,C 180.000} C_DIS
LIN {X -0.230,Y 131.236,Z 45.051,A 180.000,B 0.000,C 180.000} C_DIS
LIN {X -0.120,Y 131.236,Z 45.026,A 180.000,B 0.000,C 180.000} C_DIS
LIN {X -0.010,Y 131.236,Z 45.000,A 180.000,B 0.000,C 180.000} C_DIS
; Cutting Move Starts
LIN {X 2.498,Y 131.236,Z 45.000,A 180.000,B 0.000,C 180.000} C_DIS
LIN {X 2.500,Y 131.236,Z 52.000,A 180.000,B 0.000,C 180.000} C_DIS
LIN {X 25.181,Y 131.236,Z 52.000,A 180.000,B 0.000,C 180.000} C_DIS
LIN {X 25.181,Y 131.236,Z 57.000,A 180.000,B 0.000,C 180.000} C_DIS
LIN {X 62.700,Y 131.236,Z 57.000,A 180.000,B 0.000,C 180.000} C_DIS
LIN {X 62.701,Y 131.236,Z 62.000,A 180.000,B 0.000,C 180.000} C_DIS
LIN {X 92.299,Y 131.236,Z 62.000,A 180.000,B 0.000,C 180.000} C_DIS
LIN {X 92.299,Y 131.236,Z 57.000,A 180.000,B 0.000,C 180.000} C_DIS
LIN {X 129.818,Y 131.236,Z 57.000,A 180.000,B 0.000,C 180.000} C_DIS
LIN {X 129.819,Y 131.236,Z 52.000,A 180.000,B 0.000,C 180.000} C_DIS
LIN {X 152.500,Y 131.236,Z 52.000,A 180.000,B 0.000,C 180.000} C_DIS
LIN {X 152.500,Y 131.236,Z 45.000,A 180.000,B 0.000,C 180.000} C_DIS
LIN {X 155.010,Y 131.236,Z 45.000,A 180.000,B 0.000,C 180.000} C_DIS
; Link Move Starts
LIN {X 155.120,Y 131.236,Z 45.026,A 180.000,B 0.000,C 180.000} C_DIS
LIN {X 155.230,Y 131.236,Z 45.051,A 180.000,B 0.000,C 180.000} C_DIS
LIN {X 155.771,Y 131.549,Z 45.051,A 180.000,B 0.000,C 180.000} C_DIS
LIN {X 155.771,Y 132.174,Z 45.051,A 180.000,B 0.000,C 180.000} C_DIS
LIN {X 155.230,Y 132.486,Z 45.051,A 180.000,B 0.000,C 180.000} C_DIS
LIN {X 155.120,Y 132.486,Z 45.026,A 180.000,B 0.000,C 180.000} C_DIS
LIN {X 155.010,Y 132.486,Z 45.000,A 180.000,B 0.000,C 180.000} C_DIS
; Cutting Move Starts
LIN {X 152.500,Y 132.486,Z 45.000,A 180.000,B 0.000,C 180.000} C_DIS
LIN {X 152.500,Y 132.486,Z 52.000,A 180.000,B 0.000,C 180.000} C_DIS
LIN {X 128.503,Y 132.486,Z 52.000,A 180.000,B 0.000,C 180.000} C_DIS
LIN {X 128.502,Y 132.486,Z 57.000,A 180.000,B 0.000,C 180.000} C_DIS
LIN {X 91.049,Y 132.486,Z 57.000,A 180.000,B 0.000,C 180.000} C_DIS
LIN {X 91.049,Y 132.486,Z 62.000,A 180.000,B 0.000,C 180.000} C_DIS
LIN {X 63.951,Y 132.486,Z 62.000,A 180.000,B 0.000,C 180.000} C_DIS
LIN {X 63.951,Y 132.486,Z 57.000,A 180.000,B 0.000,C 180.000} C_DIS
LIN {X 26.497,Y 132.486,Z 57.000,A 180.000,B 0.000,C 180.000} C_DIS
LIN {X 26.497,Y 132.486,Z 52.000,A 180.000,B 0.000,C 180.000} C_DIS
LIN {X 2.500,Y 132.486,Z 52.000,A 180.000,B 0.000,C 180.000} C_DIS
LIN {X 2.498,Y 132.486,Z 45.000,A 180.000,B 0.000,C 180.000} C_DIS
LIN {X -0.010,Y 132.486,Z 45.000,A 180.000,B 0.000,C 180.000} C_DIS
; Link Move Starts
LIN {X -0.120,Y 132.486,Z 45.026,A 180.000,B 0.000,C 180.000} C_DIS
LIN {X -0.230,Y 132.486,Z 45.051,A 180.000,B 0.000,C 180.000} C_DIS
LIN {X -0.771,Y 132.799,Z 45.051,A 180.000,B 0.000,C 180.000} C_DIS
LIN {X -0.771,Y 133.423,Z 45.051,A 180.000,B 0.000,C 180.000} C_DIS
LIN {X -0.230,Y 133.736,Z 45.051,A 180.000,B 0.000,C 180.000} C_DIS
LIN {X -0.120,Y 133.736,Z 45.026,A 180.000,B 0.000,C 180.000} C_DIS
LIN {X -0.010,Y 133.736,Z 45.000,A 180.000,B 0.000,C 180.000} C_DIS
; Cutting Move Starts
LIN {X 2.500,Y 133.736,Z 45.000,A 180.000,B 0.000,C 180.000} C_DIS
LIN {X 2.500,Y 133.736,Z 52.000,A 180.000,B 0.000,C 180.000} C_DIS
LIN {X 27.880,Y 133.736,Z 52.000,A 180.000,B 0.000,C 180.000} C_DIS
LIN {X 27.880,Y 133.736,Z 57.000,A 180.000,B 0.000,C 180.000} C_DIS
LIN {X 65.200,Y 133.736,Z 57.000,A 180.000,B 0.000,C 180.000} C_DIS
LIN {X 65.200,Y 133.736,Z 62.000,A 180.000,B 0.000,C 180.000} C_DIS
LIN {X 89.800,Y 133.736,Z 62.000,A 180.000,B 0.000,C 180.000} C_DIS
LIN {X 89.800,Y 133.736,Z 57.000,A 180.000,B 0.000,C 180.000} C_DIS
LIN {X 127.120,Y 133.736,Z 57.000,A 180.000,B 0.000,C 180.000} C_DIS
LIN {X 127.120,Y 133.736,Z 52.000,A 180.000,B 0.000,C 180.000} C_DIS
LIN {X 152.500,Y 133.736,Z 52.000,A 180.000,B 0.000,C 180.000} C_DIS
LIN {X 152.500,Y 133.736,Z 45.000,A 180.000,B 0.000,C 180.000} C_DIS
LIN {X 155.010,Y 133.736,Z 45.000,A 180.000,B 0.000,C 180.000} C_DIS
; Link Move Starts
LIN {X 155.120,Y 133.736,Z 45.026,A 180.000,B 0.000,C 180.000} C_DIS
LIN {X 155.230,Y 133.736,Z 45.051,A 180.000,B 0.000,C 180.000} C_DIS
LIN {X 155.771,Y 134.048,Z 45.051,A 180.000,B 0.000,C 180.000} C_DIS
LIN {X 155.771,Y 134.673,Z 45.051,A 180.000,B 0.000,C 180.000} C_DIS
LIN {X 155.230,Y 134.986,Z 45.051,A 180.000,B 0.000,C 180.000} C_DIS
LIN {X 155.120,Y 134.986,Z 45.026,A 180.000,B 0.000,C 180.000} C_DIS
LIN {X 155.010,Y 134.986,Z 45.000,A 180.000,B 0.000,C 180.000} C_DIS
; Cutting Move Starts
LIN {X 152.500,Y 134.986,Z 45.000,A 180.000,B 0.000,C 180.000} C_DIS
LIN {X 152.500,Y 134.986,Z 52.000,A 180.000,B 0.000,C 180.000} C_DIS
LIN {X 125.664,Y 134.986,Z 52.000,A 180.000,B 0.000,C 180.000} C_DIS
LIN {X 125.664,Y 134.986,Z 57.000,A 180.000,B 0.000,C 180.000} C_DIS
LIN {X 88.550,Y 134.986,Z 57.000,A 180.000,B 0.000,C 180.000} C_DIS
LIN {X 88.550,Y 134.986,Z 62.000,A 180.000,B 0.000,C 180.000} C_DIS
LIN {X 66.450,Y 134.986,Z 62.000,A 180.000,B 0.000,C 180.000} C_DIS
LIN {X 66.450,Y 134.986,Z 57.000,A 180.000,B 0.000,C 180.000} C_DIS
LIN {X 29.335,Y 134.986,Z 57.000,A 180.000,B 0.000,C 180.000} C_DIS
LIN {X 29.335,Y 134.986,Z 52.000,A 180.000,B 0.000,C 180.000} C_DIS
LIN {X 2.500,Y 134.986,Z 52.000,A 180.000,B 0.000,C 180.000} C_DIS
LIN {X 2.500,Y 134.986,Z 45.000,A 180.000,B 0.000,C 180.000} C_DIS
LIN {X -0.010,Y 134.986,Z 45.000,A 180.000,B 0.000,C 180.000} C_DIS
; Link Move Starts
LIN {X -0.120,Y 134.986,Z 45.026,A 180.000,B 0.000,C 180.000} C_DIS
LIN {X -0.230,Y 134.986,Z 45.051,A 180.000,B 0.000,C 180.000} C_DIS
LIN {X -0.771,Y 135.298,Z 45.051,A 180.000,B 0.000,C 180.000} C_DIS
LIN {X -0.771,Y 135.923,Z 45.051,A 180.000,B 0.000,C 180.000} C_DIS
LIN {X -0.230,Y 136.236,Z 45.051,A 180.000,B 0.000,C 180.000} C_DIS
LIN {X -0.120,Y 136.236,Z 45.026,A 180.000,B 0.000,C 180.000} C_DIS
LIN {X -0.010,Y 136.236,Z 45.000,A 180.000,B 0.000,C 180.000} C_DIS
; Cutting Move Starts
LIN {X 2.500,Y 136.236,Z 45.000,A 180.000,B 0.000,C 180.000} C_DIS
LIN {X 2.500,Y 136.236,Z 52.000,A 180.000,B 0.000,C 180.000} C_DIS
LIN {X 30.869,Y 136.236,Z 52.000,A 180.000,B 0.000,C 180.000} C_DIS
LIN {X 30.869,Y 136.236,Z 57.000,A 180.000,B 0.000,C 180.000} C_DIS
LIN {X 67.700,Y 136.236,Z 57.000,A 180.000,B 0.000,C 180.000} C_DIS
LIN {X 67.700,Y 136.236,Z 62.000,A 180.000,B 0.000,C 180.000} C_DIS
LIN {X 87.300,Y 136.236,Z 62.000,A 180.000,B 0.000,C 180.000} C_DIS
LIN {X 87.300,Y 136.236,Z 57.000,A 180.000,B 0.000,C 180.000} C_DIS
LIN {X 124.131,Y 136.236,Z 57.000,A 180.000,B 0.000,C 180.000} C_DIS
LIN {X 124.131,Y 136.236,Z 52.000,A 180.000,B 0.000,C 180.000} C_DIS
LIN {X 152.500,Y 136.236,Z 52.000,A 180.000,B 0.000,C 180.000} C_DIS
LIN {X 152.500,Y 136.236,Z 45.000,A 180.000,B 0.000,C 180.000} C_DIS
LIN {X 155.010,Y 136.236,Z 45.000,A 180.000,B 0.000,C 180.000} C_DIS
; Link Move Starts
LIN {X 155.120,Y 136.236,Z 45.026,A 180.000,B 0.000,C 180.000} C_DIS
LIN {X 155.230,Y 136.236,Z 45.051,A 180.000,B 0.000,C 180.000} C_DIS
LIN {X 155.771,Y 136.548,Z 45.051,A 180.000,B 0.000,C 180.000} C_DIS
LIN {X 155.771,Y 137.173,Z 45.051,A 180.000,B 0.000,C 180.000} C_DIS
LIN {X 155.230,Y 137.486,Z 45.051,A 180.000,B 0.000,C 180.000} C_DIS
LIN {X 155.120,Y 137.486,Z 45.026,A 180.000,B 0.000,C 180.000} C_DIS
LIN {X 155.010,Y 137.486,Z 45.000,A 180.000,B 0.000,C 180.000} C_DIS
; Cutting Move Starts
LIN {X 152.500,Y 137.486,Z 45.000,A 180.000,B 0.000,C 180.000} C_DIS
LIN {X 152.500,Y 137.486,Z 52.000,A 180.000,B 0.000,C 180.000} C_DIS
LIN {X 122.511,Y 137.486,Z 52.000,A 180.000,B 0.000,C 180.000} C_DIS
LIN {X 122.511,Y 137.486,Z 57.000,A 180.000,B 0.000,C 180.000} C_DIS
LIN {X 86.050,Y 137.486,Z 57.000,A 180.000,B 0.000,C 180.000} C_DIS
LIN {X 86.050,Y 137.486,Z 62.000,A 180.000,B 0.000,C 180.000} C_DIS
LIN {X 68.950,Y 137.486,Z 62.000,A 180.000,B 0.000,C 180.000} C_DIS
LIN {X 68.950,Y 137.486,Z 57.000,A 180.000,B 0.000,C 180.000} C_DIS
LIN {X 32.489,Y 137.486,Z 57.000,A 180.000,B 0.000,C 180.000} C_DIS
LIN {X 32.489,Y 137.486,Z 52.000,A 180.000,B 0.000,C 180.000} C_DIS
LIN {X 2.500,Y 137.486,Z 52.000,A 180.000,B 0.000,C 180.000} C_DIS
LIN {X 2.500,Y 137.486,Z 45.000,A 180.000,B 0.000,C 180.000} C_DIS
LIN {X -0.010,Y 137.486,Z 45.000,A 180.000,B 0.000,C 180.000} C_DIS
; Link Move Starts
LIN {X -0.120,Y 137.486,Z 45.026,A 180.000,B 0.000,C 180.000} C_DIS
LIN {X -0.230,Y 137.486,Z 45.051,A 180.000,B 0.000,C 180.000} C_DIS
LIN {X -0.771,Y 137.798,Z 45.051,A 180.000,B 0.000,C 180.000} C_DIS
LIN {X -0.771,Y 138.423,Z 45.051,A 180.000,B 0.000,C 180.000} C_DIS
LIN {X -0.230,Y 138.736,Z 45.051,A 180.000,B 0.000,C 180.000} C_DIS
LIN {X -0.120,Y 138.736,Z 45.026,A 180.000,B 0.000,C 180.000} C_DIS
LIN {X -0.010,Y 138.736,Z 45.000,A 180.000,B 0.000,C 180.000} C_DIS
; Cutting Move Starts
LIN {X 2.500,Y 138.736,Z 45.000,A 180.000,B 0.000,C 180.000} C_DIS
LIN {X 2.500,Y 138.736,Z 52.000,A 180.000,B 0.000,C 180.000} C_DIS
LIN {X 34.203,Y 138.736,Z 52.000,A 180.000,B 0.000,C 180.000} C_DIS
LIN {X 34.203,Y 138.736,Z 57.000,A 180.000,B 0.000,C 180.000} C_DIS
LIN {X 70.199,Y 138.736,Z 57.000,A 180.000,B 0.000,C 180.000} C_DIS
LIN {X 70.200,Y 138.736,Z 62.000,A 180.000,B 0.000,C 180.000} C_DIS
LIN {X 84.800,Y 138.736,Z 62.000,A 180.000,B 0.000,C 180.000} C_DIS
LIN {X 84.800,Y 138.736,Z 57.000,A 180.000,B 0.000,C 180.000} C_DIS
LIN {X 120.797,Y 138.736,Z 57.000,A 180.000,B 0.000,C 180.000} C_DIS
LIN {X 120.797,Y 138.736,Z 52.000,A 180.000,B 0.000,C 180.000} C_DIS
LIN {X 152.500,Y 138.736,Z 52.000,A 180.000,B 0.000,C 180.000} C_DIS
LIN {X 152.500,Y 138.736,Z 45.000,A 180.000,B 0.000,C 180.000} C_DIS
LIN {X 155.010,Y 138.736,Z 45.000,A 180.000,B 0.000,C 180.000} C_DIS
; Link Move Starts
LIN {X 155.120,Y 138.736,Z 45.026,A 180.000,B 0.000,C 180.000} C_DIS
LIN {X 155.230,Y 138.736,Z 45.051,A 180.000,B 0.000,C 180.000} C_DIS
LIN {X 155.771,Y 139.048,Z 45.051,A 180.000,B 0.000,C 180.000} C_DIS
LIN {X 155.771,Y 139.673,Z 45.051,A 180.000,B 0.000,C 180.000} C_DIS
LIN {X 155.230,Y 139.985,Z 45.051,A 180.000,B 0.000,C 180.000} C_DIS
LIN {X 155.120,Y 139.985,Z 45.026,A 180.000,B 0.000,C 180.000} C_DIS
LIN {X 155.010,Y 139.985,Z 45.000,A 180.000,B 0.000,C 180.000} C_DIS
; Cutting Move Starts
LIN {X 152.500,Y 139.985,Z 45.000,A 180.000,B 0.000,C 180.000} C_DIS
LIN {X 152.500,Y 139.985,Z 52.000,A 180.000,B 0.000,C 180.000} C_DIS
LIN {X 118.980,Y 139.985,Z 52.000,A 180.000,B 0.000,C 180.000} C_DIS
LIN {X 118.980,Y 139.985,Z 57.000,A 180.000,B 0.000,C 180.000} C_DIS
LIN {X 83.550,Y 139.985,Z 57.000,A 180.000,B 0.000,C 180.000} C_DIS
LIN {X 83.549,Y 139.985,Z 62.000,A 180.000,B 0.000,C 180.000} C_DIS
LIN {X 71.450,Y 139.985,Z 62.000,A 180.000,B 0.000,C 180.000} C_DIS
LIN {X 71.450,Y 139.985,Z 57.000,A 180.000,B 0.000,C 180.000} C_DIS
LIN {X 36.020,Y 139.985,Z 57.000,A 180.000,B 0.000,C 180.000} C_DIS
LIN {X 36.019,Y 139.985,Z 52.000,A 180.000,B 0.000,C 180.000} C_DIS
LIN {X 2.500,Y 139.985,Z 52.000,A 180.000,B 0.000,C 180.000} C_DIS
LIN {X 2.500,Y 139.985,Z 45.000,A 180.000,B 0.000,C 180.000} C_DIS
LIN {X -0.010,Y 139.985,Z 45.000,A 180.000,B 0.000,C 180.000} C_DIS
; Link Move Starts
LIN {X -0.120,Y 139.985,Z 45.026,A 180.000,B 0.000,C 180.000} C_DIS
LIN {X -0.230,Y 139.985,Z 45.051,A 180.000,B 0.000,C 180.000} C_DIS
LIN {X -0.771,Y 140.298,Z 45.051,A 180.000,B 0.000,C 180.000} C_DIS
LIN {X -0.771,Y 140.923,Z 45.051,A 180.000,B 0.000,C 180.000} C_DIS
LIN {X -0.230,Y 141.235,Z 45.051,A 180.000,B 0.000,C 180.000} C_DIS
LIN {X -0.120,Y 141.235,Z 45.026,A 180.000,B 0.000,C 180.000} C_DIS
LIN {X -0.010,Y 141.235,Z 45.000,A 180.000,B 0.000,C 180.000} C_DIS
; Cutting Move Starts
LIN {X 2.497,Y 141.235,Z 45.000,A 180.000,B 0.000,C 180.000} C_DIS
LIN {X 2.500,Y 141.235,Z 52.000,A 180.000,B 0.000,C 180.000} C_DIS
LIN {X 37.976,Y 141.235,Z 52.000,A 180.000,B 0.000,C 180.000} C_DIS
LIN {X 37.976,Y 141.235,Z 57.000,A 180.000,B 0.000,C 180.000} C_DIS
LIN {X 72.700,Y 141.235,Z 57.000,A 180.000,B 0.000,C 180.000} C_DIS
LIN {X 72.700,Y 141.235,Z 62.000,A 180.000,B 0.000,C 180.000} C_DIS
LIN {X 82.298,Y 141.235,Z 62.000,A 180.000,B 0.000,C 180.000} C_DIS
LIN {X 82.300,Y 141.235,Z 57.000,A 180.000,B 0.000,C 180.000} C_DIS
LIN {X 117.024,Y 141.235,Z 57.000,A 180.000,B 0.000,C 180.000} C_DIS
LIN {X 117.024,Y 141.235,Z 52.000,A 180.000,B 0.000,C 180.000} C_DIS
LIN {X 152.500,Y 141.235,Z 52.000,A 180.000,B 0.000,C 180.000} C_DIS
LIN {X 152.500,Y 141.235,Z 45.000,A 180.000,B 0.000,C 180.000} C_DIS
LIN {X 155.010,Y 141.235,Z 45.000,A 180.000,B 0.000,C 180.000} C_DIS
; Link Move Starts
LIN {X 155.120,Y 141.235,Z 45.026,A 180.000,B 0.000,C 180.000} C_DIS
LIN {X 155.230,Y 141.235,Z 45.051,A 180.000,B 0.000,C 180.000} C_DIS
LIN {X 155.771,Y 141.548,Z 45.051,A 180.000,B 0.000,C 180.000} C_DIS
LIN {X 155.771,Y 142.173,Z 45.051,A 180.000,B 0.000,C 180.000} C_DIS
LIN {X 155.230,Y 142.485,Z 45.051,A 180.000,B 0.000,C 180.000} C_DIS
LIN {X 155.120,Y 142.485,Z 45.026,A 180.000,B 0.000,C 180.000} C_DIS
LIN {X 155.010,Y 142.485,Z 45.000,A 180.000,B 0.000,C 180.000} C_DIS
; Cutting Move Starts
LIN {X 152.500,Y 142.485,Z 45.000,A 180.000,B 0.000,C 180.000} C_DIS
LIN {X 152.500,Y 142.485,Z 52.000,A 180.000,B 0.000,C 180.000} C_DIS
LIN {X 114.934,Y 142.485,Z 52.000,A 180.000,B 0.000,C 180.000} C_DIS
LIN {X 114.934,Y 142.485,Z 57.000,A 180.000,B 0.000,C 180.000} C_DIS
LIN {X 81.050,Y 142.485,Z 57.000,A 180.000,B 0.000,C 180.000} C_DIS
LIN {X 81.049,Y 142.485,Z 62.000,A 180.000,B 0.000,C 180.000} C_DIS
LIN {X 73.950,Y 142.485,Z 62.000,A 180.000,B 0.000,C 180.000} C_DIS
LIN {X 73.949,Y 142.485,Z 57.000,A 180.000,B 0.000,C 180.000} C_DIS
LIN {X 40.066,Y 142.485,Z 57.000,A 180.000,B 0.000,C 180.000} C_DIS
LIN {X 40.065,Y 142.485,Z 52.000,A 180.000,B 0.000,C 180.000} C_DIS
LIN {X 2.500,Y 142.485,Z 52.000,A 180.000,B 0.000,C 180.000} C_DIS
LIN {X 2.500,Y 142.485,Z 45.000,A 180.000,B 0.000,C 180.000} C_DIS
LIN {X -0.010,Y 142.485,Z 45.000,A 180.000,B 0.000,C 180.000} C_DIS
; Link Move Starts
LIN {X -0.120,Y 142.485,Z 45.026,A 180.000,B 0.000,C 180.000} C_DIS
LIN {X -0.230,Y 142.485,Z 45.051,A 180.000,B 0.000,C 180.000} C_DIS
LIN {X -0.771,Y 142.798,Z 45.051,A 180.000,B 0.000,C 180.000} C_DIS
LIN {X -0.771,Y 143.423,Z 45.051,A 180.000,B 0.000,C 180.000} C_DIS
LIN {X -0.230,Y 143.735,Z 45.051,A 180.000,B 0.000,C 180.000} C_DIS
LIN {X -0.120,Y 143.735,Z 45.026,A 180.000,B 0.000,C 180.000} C_DIS
LIN {X -0.010,Y 143.735,Z 45.000,A 180.000,B 0.000,C 180.000} C_DIS
; Cutting Move Starts
LIN {X 2.499,Y 143.735,Z 45.000,A 180.000,B 0.000,C 180.000} C_DIS
LIN {X 2.500,Y 143.735,Z 52.000,A 180.000,B 0.000,C 180.000} C_DIS
LIN {X 42.322,Y 143.735,Z 52.000,A 180.000,B 0.000,C 180.000} C_DIS
LIN {X 42.322,Y 143.735,Z 57.000,A 180.000,B 0.000,C 180.000} C_DIS
LIN {X 75.200,Y 143.735,Z 57.000,A 180.000,B 0.000,C 180.000} C_DIS
LIN {X 75.200,Y 143.735,Z 62.000,A 180.000,B 0.000,C 180.000} C_DIS
LIN {X 79.800,Y 143.735,Z 62.000,A 180.000,B 0.000,C 180.000} C_DIS
LIN {X 79.800,Y 143.735,Z 57.000,A 180.000,B 0.000,C 180.000} C_DIS
LIN {X 112.677,Y 143.735,Z 57.000,A 180.000,B 0.000,C 180.000} C_DIS
LIN {X 112.678,Y 143.735,Z 52.000,A 180.000,B 0.000,C 180.000} C_DIS
LIN {X 152.500,Y 143.735,Z 52.000,A 180.000,B 0.000,C 180.000} C_DIS
LIN {X 152.500,Y 143.735,Z 45.000,A 180.000,B 0.000,C 180.000} C_DIS
LIN {X 155.010,Y 143.735,Z 45.000,A 180.000,B 0.000,C 180.000} C_DIS
; Link Move Starts
LIN {X 155.120,Y 143.735,Z 45.026,A 180.000,B 0.000,C 180.000} C_DIS
LIN {X 155.230,Y 143.735,Z 45.051,A 180.000,B 0.000,C 180.000} C_DIS
LIN {X 155.771,Y 144.048,Z 45.051,A 180.000,B 0.000,C 180.000} C_DIS
LIN {X 155.771,Y 144.673,Z 45.051,A 180.000,B 0.000,C 180.000} C_DIS
LIN {X 155.230,Y 144.985,Z 45.051,A 180.000,B 0.000,C 180.000} C_DIS
LIN {X 155.120,Y 144.985,Z 45.026,A 180.000,B 0.000,C 180.000} C_DIS
LIN {X 155.010,Y 144.985,Z 45.000,A 180.000,B 0.000,C 180.000} C_DIS
; Cutting Move Starts
LIN {X 152.500,Y 144.985,Z 45.000,A 180.000,B 0.000,C 180.000} C_DIS
LIN {X 152.500,Y 144.985,Z 52.000,A 180.000,B 0.000,C 180.000} C_DIS
LIN {X 110.214,Y 144.985,Z 52.000,A 180.000,B 0.000,C 180.000} C_DIS
LIN {X 110.213,Y 144.985,Z 57.000,A 180.000,B 0.000,C 180.000} C_DIS
LIN {X 77.773,Y 144.985,Z 57.000,A 180.000,B 0.000,C 180.000} C_DIS
LIN {X 77.773,Y 144.985,Z 62.000,A 180.000,B 0.000,C 180.000} C_DIS
LIN {X 77.227,Y 144.985,Z 62.000,A 180.000,B 0.000,C 180.000} C_DIS
LIN {X 77.222,Y 144.985,Z 57.000,A 180.000,B 0.000,C 180.000} C_DIS
LIN {X 44.786,Y 144.985,Z 57.000,A 180.000,B 0.000,C 180.000} C_DIS
LIN {X 44.786,Y 144.985,Z 52.000,A 180.000,B 0.000,C 180.000} C_DIS
LIN {X 2.500,Y 144.985,Z 52.000,A 180.000,B 0.000,C 180.000} C_DIS
LIN {X 2.500,Y 144.985,Z 45.000,A 180.000,B 0.000,C 180.000} C_DIS
LIN {X -0.010,Y 144.985,Z 45.000,A 180.000,B 0.000,C 180.000} C_DIS
; Link Move Starts
LIN {X -0.120,Y 144.985,Z 45.026,A 180.000,B 0.000,C 180.000} C_DIS
LIN {X -0.230,Y 144.985,Z 45.051,A 180.000,B 0.000,C 180.000} C_DIS
LIN {X -0.771,Y 145.298,Z 45.051,A 180.000,B 0.000,C 180.000} C_DIS
LIN {X -0.771,Y 145.922,Z 45.051,A 180.000,B 0.000,C 180.000} C_DIS
LIN {X -0.230,Y 146.235,Z 45.051,A 180.000,B 0.000,C 180.000} C_DIS
LIN {X -0.120,Y 146.235,Z 45.026,A 180.000,B 0.000,C 180.000} C_DIS
LIN {X -0.010,Y 146.235,Z 45.000,A 180.000,B 0.000,C 180.000} C_DIS
; Cutting Move Starts
LIN {X 2.500,Y 146.235,Z 45.000,A 180.000,B 0.000,C 180.000} C_DIS
LIN {X 2.500,Y 146.235,Z 52.000,A 180.000,B 0.000,C 180.000} C_DIS
LIN {X 47.502,Y 146.235,Z 52.000,A 180.000,B 0.000,C 180.000} C_DIS
LIN {X 47.504,Y 146.235,Z 57.000,A 180.000,B 0.000,C 180.000} C_DIS
LIN {X 107.496,Y 146.235,Z 57.000,A 180.000,B 0.000,C 180.000} C_DIS
LIN {X 107.496,Y 146.235,Z 52.000,A 180.000,B 0.000,C 180.000} C_DIS
LIN {X 152.500,Y 146.235,Z 52.000,A 180.000,B 0.000,C 180.000} C_DIS
LIN {X 152.500,Y 146.235,Z 45.000,A 180.000,B 0.000,C 180.000} C_DIS
LIN {X 155.010,Y 146.235,Z 45.000,A 180.000,B 0.000,C 180.000} C_DIS
; Link Move Starts
LIN {X 155.120,Y 146.235,Z 45.026,A 180.000,B 0.000,C 180.000} C_DIS
LIN {X 155.230,Y 146.235,Z 45.051,A 180.000,B 0.000,C 180.000} C_DIS
LIN {X 155.771,Y 146.547,Z 45.051,A 180.000,B 0.000,C 180.000} C_DIS
LIN {X 155.771,Y 147.172,Z 45.051,A 180.000,B 0.000,C 180.000} C_DIS
LIN {X 155.230,Y 147.485,Z 45.051,A 180.000,B 0.000,C 180.000} C_DIS
LIN {X 155.120,Y 147.485,Z 45.026,A 180.000,B 0.000,C 180.000} C_DIS
LIN {X 155.010,Y 147.485,Z 45.000,A 180.000,B 0.000,C 180.000} C_DIS
; Cutting Move Starts
LIN {X 152.500,Y 147.485,Z 45.000,A 180.000,B 0.000,C 180.000} C_DIS
LIN {X 152.500,Y 147.485,Z 52.000,A 180.000,B 0.000,C 180.000} C_DIS
LIN {X 104.453,Y 147.485,Z 52.000,A 180.000,B 0.000,C 180.000} C_DIS
LIN {X 104.453,Y 147.485,Z 57.000,A 180.000,B 0.000,C 180.000} C_DIS
LIN {X 50.547,Y 147.485,Z 57.000,A 180.000,B 0.000,C 180.000} C_DIS
LIN {X 50.547,Y 147.485,Z 52.000,A 180.000,B 0.000,C 180.000} C_DIS
LIN {X 2.500,Y 147.485,Z 52.000,A 180.000,B 0.000,C 180.000} C_DIS
LIN {X 2.500,Y 147.485,Z 45.000,A 180.000,B 0.000,C 180.000} C_DIS
LIN {X -0.010,Y 147.485,Z 45.000,A 180.000,B 0.000,C 180.000} C_DIS
; Link Move Starts
LIN {X -0.120,Y 147.485,Z 45.026,A 180.000,B 0.000,C 180.000} C_DIS
LIN {X -0.230,Y 147.485,Z 45.051,A 180.000,B 0.000,C 180.000} C_DIS
LIN {X -0.771,Y 147.797,Z 45.051,A 180.000,B 0.000,C 180.000} C_DIS
LIN {X -0.771,Y 148.422,Z 45.051,A 180.000,B 0.000,C 180.000} C_DIS
LIN {X -0.230,Y 148.735,Z 45.051,A 180.000,B 0.000,C 180.000} C_DIS
LIN {X -0.120,Y 148.735,Z 45.026,A 180.000,B 0.000,C 180.000} C_DIS
LIN {X -0.010,Y 148.735,Z 45.000,A 180.000,B 0.000,C 180.000} C_DIS
; Cutting Move Starts
LIN {X 2.500,Y 148.735,Z 45.000,A 180.000,B 0.000,C 180.000} C_DIS
LIN {X 2.500,Y 148.735,Z 52.000,A 180.000,B 0.000,C 180.000} C_DIS
LIN {X 54.051,Y 148.735,Z 52.000,A 180.000,B 0.000,C 180.000} C_DIS
LIN {X 54.051,Y 148.735,Z 57.000,A 180.000,B 0.000,C 180.000} C_DIS
LIN {X 100.949,Y 148.735,Z 57.000,A 180.000,B 0.000,C 180.000} C_DIS
LIN {X 100.949,Y 148.735,Z 52.000,A 180.000,B 0.000,C 180.000} C_DIS
LIN {X 152.500,Y 148.735,Z 52.000,A 180.000,B 0.000,C 180.000} C_DIS
LIN {X 152.500,Y 148.735,Z 45.000,A 180.000,B 0.000,C 180.000} C_DIS
LIN {X 155.010,Y 148.735,Z 45.000,A 180.000,B 0.000,C 180.000} C_DIS
; Link Move Starts
LIN {X 155.120,Y 148.735,Z 45.026,A 180.000,B 0.000,C 180.000} C_DIS
LIN {X 155.230,Y 148.735,Z 45.051,A 180.000,B 0.000,C 180.000} C_DIS
LIN {X 155.771,Y 149.047,Z 45.051,A 180.000,B 0.000,C 180.000} C_DIS
LIN {X 155.771,Y 149.672,Z 45.051,A 180.000,B 0.000,C 180.000} C_DIS
LIN {X 155.230,Y 149.985,Z 45.051,A 180.000,B 0.000,C 180.000} C_DIS
LIN {X 155.120,Y 149.985,Z 45.026,A 180.000,B 0.000,C 180.000} C_DIS
LIN {X 155.010,Y 149.985,Z 45.000,A 180.000,B 0.000,C 180.000} C_DIS
; Cutting Move Starts
LIN {X 152.500,Y 149.985,Z 45.000,A 180.000,B 0.000,C 180.000} C_DIS
LIN {X 152.500,Y 149.985,Z 52.000,A 180.000,B 0.000,C 180.000} C_DIS
LIN {X 96.756,Y 149.985,Z 52.000,A 180.000,B 0.000,C 180.000} C_DIS
LIN {X 96.756,Y 149.985,Z 57.000,A 180.000,B 0.000,C 180.000} C_DIS
LIN {X 58.244,Y 149.985,Z 57.000,A 180.000,B 0.000,C 180.000} C_DIS
LIN {X 58.244,Y 149.985,Z 52.000,A 180.000,B 0.000,C 180.000} C_DIS
LIN {X 2.500,Y 149.985,Z 52.000,A 180.000,B 0.000,C 180.000} C_DIS
LIN {X 2.500,Y 149.985,Z 45.000,A 180.000,B 0.000,C 180.000} C_DIS
LIN {X -0.010,Y 149.985,Z 45.000,A 180.000,B 0.000,C 180.000} C_DIS
; Link Move Starts
LIN {X -0.120,Y 149.985,Z 45.026,A 180.000,B 0.000,C 180.000} C_DIS
LIN {X -0.230,Y 149.985,Z 45.051,A 180.000,B 0.000,C 180.000} C_DIS
LIN {X -0.771,Y 150.297,Z 45.051,A 180.000,B 0.000,C 180.000} C_DIS
LIN {X -0.771,Y 150.922,Z 45.051,A 180.000,B 0.000,C 180.000} C_DIS
LIN {X -0.230,Y 151.235,Z 45.051,A 180.000,B 0.000,C 180.000} C_DIS
LIN {X -0.120,Y 151.235,Z 45.026,A 180.000,B 0.000,C 180.000} C_DIS
LIN {X -0.010,Y 151.235,Z 45.000,A 180.000,B 0.000,C 180.000} C_DIS
; Cutting Move Starts
LIN {X 2.826,Y 151.235,Z 45.000,A 180.000,B 0.000,C 180.000} C_DIS
LIN {X 2.826,Y 151.235,Z 52.000,A 180.000,B 0.000,C 180.000} C_DIS
LIN {X 63.795,Y 151.235,Z 52.000,A 180.000,B 0.000,C 180.000} C_DIS
LIN {X 63.795,Y 151.235,Z 57.000,A 180.000,B 0.000,C 180.000} C_DIS
LIN {X 91.205,Y 151.235,Z 57.000,A 180.000,B 0.000,C 180.000} C_DIS
LIN {X 91.205,Y 151.235,Z 52.000,A 180.000,B 0.000,C 180.000} C_DIS
LIN {X 152.174,Y 151.235,Z 52.000,A 180.000,B 0.000,C 180.000} C_DIS
LIN {X 152.174,Y 151.235,Z 45.000,A 180.000,B 0.000,C 180.000} C_DIS
LIN {X 155.010,Y 151.235,Z 45.000,A 180.000,B 0.000,C 180.000} C_DIS
; Link Move Starts
LIN {X 155.120,Y 151.235,Z 45.026,A 180.000,B 0.000,C 180.000} C_DIS
LIN {X 155.230,Y 151.235,Z 45.051,A 180.000,B 0.000,C 180.000} C_DIS
LIN {X 155.771,Y 151.547,Z 45.051,A 180.000,B 0.000,C 180.000} C_DIS
LIN {X 155.771,Y 152.172,Z 45.051,A 180.000,B 0.000,C 180.000} C_DIS
LIN {X 155.230,Y 152.484,Z 45.051,A 180.000,B 0.000,C 180.000} C_DIS
LIN {X 155.120,Y 152.484,Z 45.026,A 180.000,B 0.000,C 180.000} C_DIS
LIN {X 155.010,Y 152.484,Z 45.000,A 180.000,B 0.000,C 180.000} C_DIS
; Cutting Move Starts
LIN {X 150.279,Y 152.484,Z 45.000,A 180.000,B 0.000,C 180.000} C_DIS
LIN {X 150.279,Y 152.484,Z 52.000,A 180.000,B 0.000,C 180.000} C_DIS
LIN {X 78.843,Y 152.484,Z 52.000,A 180.000,B 0.000,C 180.000} C_DIS
LIN {X 78.843,Y 152.484,Z 57.000,A 180.000,B 0.000,C 180.000} C_DIS
LIN {X 76.157,Y 152.484,Z 57.000,A 180.000,B 0.000,C 180.000} C_DIS
LIN {X 76.157,Y 152.484,Z 52.000,A 180.000,B 0.000,C 180.000} C_DIS
LIN {X 4.721,Y 152.484,Z 52.000,A 180.000,B 0.000,C 180.000} C_DIS
LIN {X 4.721,Y 152.484,Z 45.000,A 180.000,B 0.000,C 180.000} C_DIS
LIN {X -0.010,Y 152.484,Z 45.000,A 180.000,B 0.000,C 180.000} C_DIS
; Link Move Starts
LIN {X -0.120,Y 152.484,Z 45.026,A 180.000,B 0.000,C 180.000} C_DIS
LIN {X -0.230,Y 152.484,Z 45.051,A 180.000,B 0.000,C 180.000} C_DIS
LIN {X -0.771,Y 152.797,Z 45.051,A 180.000,B 0.000,C 180.000} C_DIS
LIN {X -0.771,Y 153.422,Z 45.051,A 180.000,B 0.000,C 180.000} C_DIS
LIN {X -0.230,Y 153.734,Z 45.051,A 180.000,B 0.000,C 180.000} C_DIS
LIN {X -0.120,Y 153.734,Z 45.026,A 180.000,B 0.000,C 180.000} C_DIS
LIN {X -0.010,Y 153.734,Z 45.000,A 180.000,B 0.000,C 180.000} C_DIS
; Cutting Move Starts
LIN {X 155.010,Y 153.734,Z 45.000,A 180.000,B 0.000,C 180.000} C_DIS
; Link Move Starts
LIN {X 155.120,Y 153.734,Z 45.026,A 180.000,B 0.000,C 180.000} C_DIS
LIN {X 155.230,Y 153.734,Z 45.051,A 180.000,B 0.000,C 180.000} C_DIS
LIN {X 155.771,Y 154.047,Z 45.051,A 180.000,B 0.000,C 180.000} C_DIS
LIN {X 155.771,Y 154.672,Z 45.051,A 180.000,B 0.000,C 180.000} C_DIS
LIN {X 155.230,Y 154.984,Z 45.051,A 180.000,B 0.000,C 180.000} C_DIS
LIN {X 155.120,Y 154.984,Z 45.026,A 180.000,B 0.000,C 180.000} C_DIS
LIN {X 155.010,Y 154.984,Z 45.000,A 180.000,B 0.000,C 180.000} C_DIS
; Cutting Move Starts
LIN {X -0.010,Y 154.984,Z 45.000,A 180.000,B 0.000,C 180.000} C_DIS
; Lead Out Move Starts
LIN {X -0.363,Y 154.984,Z 45.146,A 180.000,B 0.000,C 180.000} C_DIS
LIN {X -0.510,Y 154.984,Z 45.500,A 180.000,B 0.000,C 180.000} C_DIS
; Rapid Move Starts
LIN {X -0.510,Y 154.984,Z 105.000,A 180.000,B 0.000,C 180.000} C_DIS
;ENDFOLD
END

--- sParallel2.dat ---
&ACCESS RVO
DEFDAT sParallel2
;FOLD EXTERNAL DECLARATIONS;%{PE}%MKUKATPBASIS,%CEXT,%VCOMMON,%P
  ;FOLD BASISTECH EXT;%{PE}%MKUKATPBASIS,%CEXT,%VEXT,%P
    EXT  BAS (BAS_COMMAND  :IN,REAL  :IN )
  ;ENDFOLD (BASISTECH EXT)

;ENDFOLD (EXTERNAL DECLARATIONS)
ENDDAT
